   STATUS[676].EXT.BIT30 := FALSE;
   STATUS[676].EXT.BIT31 := FALSE;
   STATUS[676].EXT.ModeBit1 := FALSE;
   STATUS[676].EXT.ModeBit2 := FALSE;
   STATUS[676].EXT.ModeBit3 := FALSE;
   STATUS[676].EXT.BIT19 := FALSE;
   STATUS[676].EXT.BIT20 := FALSE;
   STATUS[676].EXT.AlarmSuppressed := FALSE;
   STATUS[676].EXT.AlarmPresent := FALSE;
   STATUS[676].EXT.AlarmFailUnAck := FALSE;
   STATUS[676].Status := 0;
   STATUS[676].TimeStamp := 16#0000;
   STATUS[677].EXT.AlarmWarnUnAck := FALSE;
   STATUS[677].EXT.AckRequired := FALSE;
   STATUS[677].EXT.Maintanence := FALSE;
   STATUS[677].EXT.Operation := FALSE;
   STATUS[677].EXT.Forced := FALSE;
   STATUS[677].EXT.BIT29 := FALSE;
   STATUS[677].EXT.BIT30 := FALSE;
   STATUS[677].EXT.BIT31 := FALSE;
   STATUS[677].EXT.ModeBit1 := FALSE;
   STATUS[677].EXT.ModeBit2 := FALSE;
   STATUS[677].EXT.ModeBit3 := FALSE;
   STATUS[677].EXT.BIT19 := FALSE;
   STATUS[677].EXT.BIT20 := FALSE;
   STATUS[677].EXT.AlarmSuppressed := FALSE;
   STATUS[677].EXT.AlarmPresent := FALSE;
   STATUS[677].EXT.AlarmFailUnAck := FALSE;
   STATUS[677].Status := 0;
   STATUS[677].TimeStamp := 16#0000;
   STATUS[678].EXT.AlarmWarnUnAck := FALSE;
   STATUS[678].EXT.AckRequired := FALSE;
   STATUS[678].EXT.Maintanence := FALSE;
   STATUS[678].EXT.Operation := FALSE;
   STATUS[678].EXT.Forced := FALSE;
   STATUS[678].EXT.BIT29 := FALSE;
   STATUS[678].EXT.BIT30 := FALSE;
   STATUS[678].EXT.BIT31 := FALSE;
   STATUS[678].EXT.ModeBit1 := FALSE;
   STATUS[678].EXT.ModeBit2 := FALSE;
   STATUS[678].EXT.ModeBit3 := FALSE;
   STATUS[678].EXT.BIT19 := FALSE;
   STATUS[678].EXT.BIT20 := FALSE;
   STATUS[678].EXT.AlarmSuppressed := FALSE;
   STATUS[678].EXT.AlarmPresent := FALSE;
   STATUS[678].EXT.AlarmFailUnAck := FALSE;
   STATUS[678].Status := 0;
   STATUS[678].TimeStamp := 16#0000;
   STATUS[679].EXT.AlarmWarnUnAck := FALSE;
   STATUS[679].EXT.AckRequired := FALSE;
   STATUS[679].EXT.Maintanence := FALSE;
   STATUS[679].EXT.Operation := FALSE;
   STATUS[679].EXT.Forced := FALSE;
   STATUS[679].EXT.BIT29 := FALSE;
   STATUS[679].EXT.BIT30 := FALSE;
   STATUS[679].EXT.BIT31 := FALSE;
   STATUS[679].EXT.ModeBit1 := FALSE;
   STATUS[679].EXT.ModeBit2 := FALSE;
   STATUS[679].EXT.ModeBit3 := FALSE;
   STATUS[679].EXT.BIT19 := FALSE;
   STATUS[679].EXT.BIT20 := FALSE;
   STATUS[679].EXT.AlarmSuppressed := FALSE;
   STATUS[679].EXT.AlarmPresent := FALSE;
   STATUS[679].EXT.AlarmFailUnAck := FALSE;
   STATUS[679].Status := 0;
   STATUS[679].TimeStamp := 16#0000;
   STATUS[680].EXT.AlarmWarnUnAck := FALSE;
   STATUS[680].EXT.AckRequired := FALSE;
   STATUS[680].EXT.Maintanence := FALSE;
   STATUS[680].EXT.Operation := FALSE;
   STATUS[680].EXT.Forced := FALSE;
   STATUS[680].EXT.BIT29 := FALSE;
   STATUS[680].EXT.BIT30 := FALSE;
   STATUS[680].EXT.BIT31 := FALSE;
   STATUS[680].EXT.ModeBit1 := FALSE;
   STATUS[680].EXT.ModeBit2 := FALSE;
   STATUS[680].EXT.ModeBit3 := FALSE;
   STATUS[680].EXT.BIT19 := FALSE;
   STATUS[680].EXT.BIT20 := FALSE;
   STATUS[680].EXT.AlarmSuppressed := FALSE;
   STATUS[680].EXT.AlarmPresent := FALSE;
   STATUS[680].EXT.AlarmFailUnAck := FALSE;
   STATUS[680].Status := 0;
   STATUS[680].TimeStamp := 16#0000;
   STATUS[681].EXT.AlarmWarnUnAck := FALSE;
   STATUS[681].EXT.AckRequired := FALSE;
   STATUS[681].EXT.Maintanence := FALSE;
   STATUS[681].EXT.Operation := FALSE;
   STATUS[681].EXT.Forced := FALSE;
   STATUS[681].EXT.BIT29 := FALSE;
   STATUS[681].EXT.BIT30 := FALSE;
   STATUS[681].EXT.BIT31 := FALSE;
   STATUS[681].EXT.ModeBit1 := FALSE;
   STATUS[681].EXT.ModeBit2 := FALSE;
   STATUS[681].EXT.ModeBit3 := FALSE;
   STATUS[681].EXT.BIT19 := FALSE;
   STATUS[681].EXT.BIT20 := FALSE;
   STATUS[681].EXT.AlarmSuppressed := FALSE;
   STATUS[681].EXT.AlarmPresent := FALSE;
   STATUS[681].EXT.AlarmFailUnAck := FALSE;
   STATUS[681].Status := 0;
   STATUS[681].TimeStamp := 16#0000;
   STATUS[682].EXT.AlarmWarnUnAck := FALSE;
   STATUS[682].EXT.AckRequired := FALSE;
   STATUS[682].EXT.Maintanence := FALSE;
   STATUS[682].EXT.Operation := FALSE;
   STATUS[682].EXT.Forced := FALSE;
   STATUS[682].EXT.BIT29 := FALSE;
   STATUS[682].EXT.BIT30 := FALSE;
   STATUS[682].EXT.BIT31 := FALSE;
   STATUS[682].EXT.ModeBit1 := FALSE;
   STATUS[682].EXT.ModeBit2 := FALSE;
   STATUS[682].EXT.ModeBit3 := FALSE;
   STATUS[682].EXT.BIT19 := FALSE;
   STATUS[682].EXT.BIT20 := FALSE;
   STATUS[682].EXT.AlarmSuppressed := FALSE;
   STATUS[682].EXT.AlarmPresent := FALSE;
   STATUS[682].EXT.AlarmFailUnAck := FALSE;
   STATUS[682].Status := 0;
   STATUS[682].TimeStamp := 16#0000;
   STATUS[683].EXT.AlarmWarnUnAck := FALSE;
   STATUS[683].EXT.AckRequired := FALSE;
   STATUS[683].EXT.Maintanence := FALSE;
   STATUS[683].EXT.Operation := FALSE;
   STATUS[683].EXT.Forced := FALSE;
   STATUS[683].EXT.BIT29 := FALSE;
   STATUS[683].EXT.BIT30 := FALSE;
   STATUS[683].EXT.BIT31 := FALSE;
   STATUS[683].EXT.ModeBit1 := FALSE;
   STATUS[683].EXT.ModeBit2 := FALSE;
   STATUS[683].EXT.ModeBit3 := FALSE;
   STATUS[683].EXT.BIT19 := FALSE;
   STATUS[683].EXT.BIT20 := FALSE;
   STATUS[683].EXT.AlarmSuppressed := FALSE;
   STATUS[683].EXT.AlarmPresent := FALSE;
   STATUS[683].EXT.AlarmFailUnAck := FALSE;
   STATUS[683].Status := 0;
   STATUS[683].TimeStamp := 16#0000;
   STATUS[684].EXT.AlarmWarnUnAck := FALSE;
   STATUS[684].EXT.AckRequired := FALSE;
   STATUS[684].EXT.Maintanence := FALSE;
   STATUS[684].EXT.Operation := FALSE;
   STATUS[684].EXT.Forced := FALSE;
   STATUS[684].EXT.BIT29 := FALSE;
   STATUS[684].EXT.BIT30 := FALSE;
   STATUS[684].EXT.BIT31 := FALSE;
   STATUS[684].EXT.ModeBit1 := FALSE;
   STATUS[684].EXT.ModeBit2 := FALSE;
   STATUS[684].EXT.ModeBit3 := FALSE;
   STATUS[684].EXT.BIT19 := FALSE;
   STATUS[684].EXT.BIT20 := FALSE;
   STATUS[684].EXT.AlarmSuppressed := FALSE;
   STATUS[684].EXT.AlarmPresent := FALSE;
   STATUS[684].EXT.AlarmFailUnAck := FALSE;
   STATUS[684].Status := 0;
   STATUS[684].TimeStamp := 16#0000;
   STATUS[685].EXT.AlarmWarnUnAck := FALSE;
   STATUS[685].EXT.AckRequired := FALSE;
   STATUS[685].EXT.Maintanence := FALSE;
   STATUS[685].EXT.Operation := FALSE;
   STATUS[685].EXT.Forced := FALSE;
   STATUS[685].EXT.BIT29 := FALSE;
   STATUS[685].EXT.BIT30 := FALSE;
   STATUS[685].EXT.BIT31 := FALSE;
   STATUS[685].EXT.ModeBit1 := FALSE;
   STATUS[685].EXT.ModeBit2 := FALSE;
   STATUS[685].EXT.ModeBit3 := FALSE;
   STATUS[685].EXT.BIT19 := FALSE;
   STATUS[685].EXT.BIT20 := FALSE;
   STATUS[685].EXT.AlarmSuppressed := FALSE;
   STATUS[685].EXT.AlarmPresent := FALSE;
   STATUS[685].EXT.AlarmFailUnAck := FALSE;
   STATUS[685].Status := 0;
   STATUS[685].TimeStamp := 16#0000;
   STATUS[686].EXT.AlarmWarnUnAck := FALSE;
   STATUS[686].EXT.AckRequired := FALSE;
   STATUS[686].EXT.Maintanence := FALSE;
   STATUS[686].EXT.Operation := FALSE;
   STATUS[686].EXT.Forced := FALSE;
   STATUS[686].EXT.BIT29 := FALSE;
   STATUS[686].EXT.BIT30 := FALSE;
   STATUS[686].EXT.BIT31 := FALSE;
   STATUS[686].EXT.ModeBit1 := FALSE;
   STATUS[686].EXT.ModeBit2 := FALSE;
   STATUS[686].EXT.ModeBit3 := FALSE;
   STATUS[686].EXT.BIT19 := FALSE;
   STATUS[686].EXT.BIT20 := FALSE;
   STATUS[686].EXT.AlarmSuppressed := FALSE;
   STATUS[686].EXT.AlarmPresent := FALSE;
   STATUS[686].EXT.AlarmFailUnAck := FALSE;
   STATUS[686].Status := 0;
   STATUS[686].TimeStamp := 16#0000;
   STATUS[687].EXT.AlarmWarnUnAck := FALSE;
   STATUS[687].EXT.AckRequired := FALSE;
   STATUS[687].EXT.Maintanence := FALSE;
   STATUS[687].EXT.Operation := FALSE;
   STATUS[687].EXT.Forced := FALSE;
   STATUS[687].EXT.BIT29 := FALSE;
   STATUS[687].EXT.BIT30 := FALSE;
   STATUS[687].EXT.BIT31 := FALSE;
   STATUS[687].EXT.ModeBit1 := FALSE;
   STATUS[687].EXT.ModeBit2 := FALSE;
   STATUS[687].EXT.ModeBit3 := FALSE;
   STATUS[687].EXT.BIT19 := FALSE;
   STATUS[687].EXT.BIT20 := FALSE;
   STATUS[687].EXT.AlarmSuppressed := FALSE;
   STATUS[687].EXT.AlarmPresent := FALSE;
   STATUS[687].EXT.AlarmFailUnAck := FALSE;
   STATUS[687].Status := 0;
   STATUS[687].TimeStamp := 16#0000;
   STATUS[688].EXT.AlarmWarnUnAck := FALSE;
   STATUS[688].EXT.AckRequired := FALSE;
   STATUS[688].EXT.Maintanence := FALSE;
   STATUS[688].EXT.Operation := FALSE;
   STATUS[688].EXT.Forced := FALSE;
   STATUS[688].EXT.BIT29 := FALSE;
   STATUS[688].EXT.BIT30 := FALSE;
   STATUS[688].EXT.BIT31 := FALSE;
   STATUS[688].EXT.ModeBit1 := FALSE;
   STATUS[688].EXT.ModeBit2 := FALSE;
   STATUS[688].EXT.ModeBit3 := FALSE;
   STATUS[688].EXT.BIT19 := FALSE;
   STATUS[688].EXT.BIT20 := FALSE;
   STATUS[688].EXT.AlarmSuppressed := FALSE;
   STATUS[688].EXT.AlarmPresent := FALSE;
   STATUS[688].EXT.AlarmFailUnAck := FALSE;
   STATUS[688].Status := 0;
   STATUS[688].TimeStamp := 16#0000;
   STATUS[689].EXT.AlarmWarnUnAck := FALSE;
   STATUS[689].EXT.AckRequired := FALSE;
   STATUS[689].EXT.Maintanence := FALSE;
   STATUS[689].EXT.Operation := FALSE;
   STATUS[689].EXT.Forced := FALSE;
   STATUS[689].EXT.BIT29 := FALSE;
   STATUS[689].EXT.BIT30 := FALSE;
   STATUS[689].EXT.BIT31 := FALSE;
   STATUS[689].EXT.ModeBit1 := FALSE;
   STATUS[689].EXT.ModeBit2 := FALSE;
   STATUS[689].EXT.ModeBit3 := FALSE;
   STATUS[689].EXT.BIT19 := FALSE;
   STATUS[689].EXT.BIT20 := FALSE;
   STATUS[689].EXT.AlarmSuppressed := FALSE;
   STATUS[689].EXT.AlarmPresent := FALSE;
   STATUS[689].EXT.AlarmFailUnAck := FALSE;
   STATUS[689].Status := 0;
   STATUS[689].TimeStamp := 16#0000;
   STATUS[690].EXT.AlarmWarnUnAck := FALSE;
   STATUS[690].EXT.AckRequired := FALSE;
   STATUS[690].EXT.Maintanence := FALSE;
   STATUS[690].EXT.Operation := FALSE;
   STATUS[690].EXT.Forced := FALSE;
   STATUS[690].EXT.BIT29 := FALSE;
   STATUS[690].EXT.BIT30 := FALSE;
   STATUS[690].EXT.BIT31 := FALSE;
   STATUS[690].EXT.ModeBit1 := FALSE;
   STATUS[690].EXT.ModeBit2 := FALSE;
   STATUS[690].EXT.ModeBit3 := FALSE;
   STATUS[690].EXT.BIT19 := FALSE;
   STATUS[690].EXT.BIT20 := FALSE;
   STATUS[690].EXT.AlarmSuppressed := FALSE;
   STATUS[690].EXT.AlarmPresent := FALSE;
   STATUS[690].EXT.AlarmFailUnAck := FALSE;
   STATUS[690].Status := 0;
   STATUS[690].TimeStamp := 16#0000;
   STATUS[691].EXT.AlarmWarnUnAck := FALSE;
   STATUS[691].EXT.AckRequired := FALSE;
   STATUS[691].EXT.Maintanence := FALSE;
   STATUS[691].EXT.Operation := FALSE;
   STATUS[691].EXT.Forced := FALSE;
   STATUS[691].EXT.BIT29 := FALSE;
   STATUS[691].EXT.BIT30 := FALSE;
   STATUS[691].EXT.BIT31 := FALSE;
   STATUS[691].EXT.ModeBit1 := FALSE;
   STATUS[691].EXT.ModeBit2 := FALSE;
   STATUS[691].EXT.ModeBit3 := FALSE;
   STATUS[691].EXT.BIT19 := FALSE;
   STATUS[691].EXT.BIT20 := FALSE;
   STATUS[691].EXT.AlarmSuppressed := FALSE;
   STATUS[691].EXT.AlarmPresent := FALSE;
   STATUS[691].EXT.AlarmFailUnAck := FALSE;
   STATUS[691].Status := 0;
   STATUS[691].TimeStamp := 16#0000;
   STATUS[692].EXT.AlarmWarnUnAck := FALSE;
   STATUS[692].EXT.AckRequired := FALSE;
   STATUS[692].EXT.Maintanence := FALSE;
   STATUS[692].EXT.Operation := FALSE;
   STATUS[692].EXT.Forced := FALSE;
   STATUS[692].EXT.BIT29 := FALSE;
   STATUS[692].EXT.BIT30 := FALSE;
   STATUS[692].EXT.BIT31 := FALSE;
   STATUS[692].EXT.ModeBit1 := FALSE;
   STATUS[692].EXT.ModeBit2 := FALSE;
   STATUS[692].EXT.ModeBit3 := FALSE;
   STATUS[692].EXT.BIT19 := FALSE;
   STATUS[692].EXT.BIT20 := FALSE;
   STATUS[692].EXT.AlarmSuppressed := FALSE;
   STATUS[692].EXT.AlarmPresent := FALSE;
   STATUS[692].EXT.AlarmFailUnAck := FALSE;
   STATUS[692].Status := 0;
   STATUS[692].TimeStamp := 16#0000;
   STATUS[693].EXT.AlarmWarnUnAck := FALSE;
   STATUS[693].EXT.AckRequired := FALSE;
   STATUS[693].EXT.Maintanence := FALSE;
   STATUS[693].EXT.Operation := FALSE;
   STATUS[693].EXT.Forced := FALSE;
   STATUS[693].EXT.BIT29 := FALSE;
   STATUS[693].EXT.BIT30 := FALSE;
   STATUS[693].EXT.BIT31 := FALSE;
   STATUS[693].EXT.ModeBit1 := FALSE;
   STATUS[693].EXT.ModeBit2 := FALSE;
   STATUS[693].EXT.ModeBit3 := FALSE;
   STATUS[693].EXT.BIT19 := FALSE;
   STATUS[693].EXT.BIT20 := FALSE;
   STATUS[693].EXT.AlarmSuppressed := FALSE;
   STATUS[693].EXT.AlarmPresent := FALSE;
   STATUS[693].EXT.AlarmFailUnAck := FALSE;
   STATUS[693].Status := 0;
   STATUS[693].TimeStamp := 16#0000;
   STATUS[694].EXT.AlarmWarnUnAck := FALSE;
   STATUS[694].EXT.AckRequired := FALSE;
   STATUS[694].EXT.Maintanence := FALSE;
   STATUS[694].EXT.Operation := FALSE;
   STATUS[694].EXT.Forced := FALSE;
   STATUS[694].EXT.BIT29 := FALSE;
   STATUS[694].EXT.BIT30 := FALSE;
   STATUS[694].EXT.BIT31 := FALSE;
   STATUS[694].EXT.ModeBit1 := FALSE;
   STATUS[694].EXT.ModeBit2 := FALSE;
   STATUS[694].EXT.ModeBit3 := FALSE;
   STATUS[694].EXT.BIT19 := FALSE;
   STATUS[694].EXT.BIT20 := FALSE;
   STATUS[694].EXT.AlarmSuppressed := FALSE;
   STATUS[694].EXT.AlarmPresent := FALSE;
   STATUS[694].EXT.AlarmFailUnAck := FALSE;
   STATUS[694].Status := 0;
   STATUS[694].TimeStamp := 16#0000;
   STATUS[695].EXT.AlarmWarnUnAck := FALSE;
   STATUS[695].EXT.AckRequired := FALSE;
   STATUS[695].EXT.Maintanence := FALSE;
   STATUS[695].EXT.Operation := FALSE;
   STATUS[695].EXT.Forced := FALSE;
   STATUS[695].EXT.BIT29 := FALSE;
   STATUS[695].EXT.BIT30 := FALSE;
   STATUS[695].EXT.BIT31 := FALSE;
   STATUS[695].EXT.ModeBit1 := FALSE;
   STATUS[695].EXT.ModeBit2 := FALSE;
   STATUS[695].EXT.ModeBit3 := FALSE;
   STATUS[695].EXT.BIT19 := FALSE;
   STATUS[695].EXT.BIT20 := FALSE;
   STATUS[695].EXT.AlarmSuppressed := FALSE;
   STATUS[695].EXT.AlarmPresent := FALSE;
   STATUS[695].EXT.AlarmFailUnAck := FALSE;
   STATUS[695].Status := 0;
   STATUS[695].TimeStamp := 16#0000;
   STATUS[696].EXT.AlarmWarnUnAck := FALSE;
   STATUS[696].EXT.AckRequired := FALSE;
   STATUS[696].EXT.Maintanence := FALSE;
   STATUS[696].EXT.Operation := FALSE;
   STATUS[696].EXT.Forced := FALSE;
   STATUS[696].EXT.BIT29 := FALSE;
   STATUS[696].EXT.BIT30 := FALSE;
   STATUS[696].EXT.BIT31 := FALSE;
   STATUS[696].EXT.ModeBit1 := FALSE;
   STATUS[696].EXT.ModeBit2 := FALSE;
   STATUS[696].EXT.ModeBit3 := FALSE;
   STATUS[696].EXT.BIT19 := FALSE;
   STATUS[696].EXT.BIT20 := FALSE;
   STATUS[696].EXT.AlarmSuppressed := FALSE;
   STATUS[696].EXT.AlarmPresent := FALSE;
   STATUS[696].EXT.AlarmFailUnAck := FALSE;
   STATUS[696].Status := 0;
   STATUS[696].TimeStamp := 16#0000;
   STATUS[697].EXT.AlarmWarnUnAck := FALSE;
   STATUS[697].EXT.AckRequired := FALSE;
   STATUS[697].EXT.Maintanence := FALSE;
   STATUS[697].EXT.Operation := FALSE;
   STATUS[697].EXT.Forced := FALSE;
   STATUS[697].EXT.BIT29 := FALSE;
   STATUS[697].EXT.BIT30 := FALSE;
   STATUS[697].EXT.BIT31 := FALSE;
   STATUS[697].EXT.ModeBit1 := FALSE;
   STATUS[697].EXT.ModeBit2 := FALSE;
   STATUS[697].EXT.ModeBit3 := FALSE;
   STATUS[697].EXT.BIT19 := FALSE;
   STATUS[697].EXT.BIT20 := FALSE;
   STATUS[697].EXT.AlarmSuppressed := FALSE;
   STATUS[697].EXT.AlarmPresent := FALSE;
   STATUS[697].EXT.AlarmFailUnAck := FALSE;
   STATUS[697].Status := 0;
   STATUS[697].TimeStamp := 16#0000;
   STATUS[698].EXT.AlarmWarnUnAck := FALSE;
   STATUS[698].EXT.AckRequired := FALSE;
   STATUS[698].EXT.Maintanence := FALSE;
   STATUS[698].EXT.Operation := FALSE;
   STATUS[698].EXT.Forced := FALSE;
   STATUS[698].EXT.BIT29 := FALSE;
   STATUS[698].EXT.BIT30 := FALSE;
   STATUS[698].EXT.BIT31 := FALSE;
   STATUS[698].EXT.ModeBit1 := FALSE;
   STATUS[698].EXT.ModeBit2 := FALSE;
   STATUS[698].EXT.ModeBit3 := FALSE;
   STATUS[698].EXT.BIT19 := FALSE;
   STATUS[698].EXT.BIT20 := FALSE;
   STATUS[698].EXT.AlarmSuppressed := FALSE;
   STATUS[698].EXT.AlarmPresent := FALSE;
   STATUS[698].EXT.AlarmFailUnAck := FALSE;
   STATUS[698].Status := 0;
   STATUS[698].TimeStamp := 16#0000;
   STATUS[699].EXT.AlarmWarnUnAck := FALSE;
   STATUS[699].EXT.AckRequired := FALSE;
   STATUS[699].EXT.Maintanence := FALSE;
   STATUS[699].EXT.Operation := FALSE;
   STATUS[699].EXT.Forced := FALSE;
   STATUS[699].EXT.BIT29 := FALSE;
   STATUS[699].EXT.BIT30 := FALSE;
   STATUS[699].EXT.BIT31 := FALSE;
   STATUS[699].EXT.ModeBit1 := FALSE;
   STATUS[699].EXT.ModeBit2 := FALSE;
   STATUS[699].EXT.ModeBit3 := FALSE;
   STATUS[699].EXT.BIT19 := FALSE;
   STATUS[699].EXT.BIT20 := FALSE;
   STATUS[699].EXT.AlarmSuppressed := FALSE;
   STATUS[699].EXT.AlarmPresent := FALSE;
   STATUS[699].EXT.AlarmFailUnAck := FALSE;
   STATUS[699].Status := 0;
   STATUS[699].TimeStamp := 16#0000;
   STATUS[700].EXT.AlarmWarnUnAck := FALSE;
   STATUS[700].EXT.AckRequired := FALSE;
   STATUS[700].EXT.Maintanence := FALSE;
   STATUS[700].EXT.Operation := FALSE;
   STATUS[700].EXT.Forced := FALSE;
   STATUS[700].EXT.BIT29 := FALSE;
   STATUS[700].EXT.BIT30 := FALSE;
   STATUS[700].EXT.BIT31 := FALSE;
   STATUS[700].EXT.ModeBit1 := FALSE;
   STATUS[700].EXT.ModeBit2 := FALSE;
   STATUS[700].EXT.ModeBit3 := FALSE;
   STATUS[700].EXT.BIT19 := FALSE;
   STATUS[700].EXT.BIT20 := FALSE;
   STATUS[700].EXT.AlarmSuppressed := FALSE;
   STATUS[700].EXT.AlarmPresent := FALSE;
   STATUS[700].EXT.AlarmFailUnAck := FALSE;
   STATUS[700].Status := 0;
   STATUS[700].TimeStamp := 16#0000;
   STATUS[701].EXT.AlarmWarnUnAck := FALSE;
   STATUS[701].EXT.AckRequired := FALSE;
   STATUS[701].EXT.Maintanence := FALSE;
   STATUS[701].EXT.Operation := FALSE;
   STATUS[701].EXT.Forced := FALSE;
   STATUS[701].EXT.BIT29 := FALSE;
   STATUS[701].EXT.BIT30 := FALSE;
   STATUS[701].EXT.BIT31 := FALSE;
   STATUS[701].EXT.ModeBit1 := FALSE;
   STATUS[701].EXT.ModeBit2 := FALSE;
   STATUS[701].EXT.ModeBit3 := FALSE;
   STATUS[701].EXT.BIT19 := FALSE;
   STATUS[701].EXT.BIT20 := FALSE;
   STATUS[701].EXT.AlarmSuppressed := FALSE;
   STATUS[701].EXT.AlarmPresent := FALSE;
   STATUS[701].EXT.AlarmFailUnAck := FALSE;
   STATUS[701].Status := 0;
   STATUS[701].TimeStamp := 16#0000;
   STATUS[702].EXT.AlarmWarnUnAck := FALSE;
   STATUS[702].EXT.AckRequired := FALSE;
   STATUS[702].EXT.Maintanence := FALSE;
   STATUS[702].EXT.Operation := FALSE;
   STATUS[702].EXT.Forced := FALSE;
   STATUS[702].EXT.BIT29 := FALSE;
   STATUS[702].EXT.BIT30 := FALSE;
   STATUS[702].EXT.BIT31 := FALSE;
   STATUS[702].EXT.ModeBit1 := FALSE;
   STATUS[702].EXT.ModeBit2 := FALSE;
   STATUS[702].EXT.ModeBit3 := FALSE;
   STATUS[702].EXT.BIT19 := FALSE;
   STATUS[702].EXT.BIT20 := FALSE;
   STATUS[702].EXT.AlarmSuppressed := FALSE;
   STATUS[702].EXT.AlarmPresent := FALSE;
   STATUS[702].EXT.AlarmFailUnAck := FALSE;
   STATUS[702].Status := 0;
   STATUS[702].TimeStamp := 16#0000;
   STATUS[703].EXT.AlarmWarnUnAck := FALSE;
   STATUS[703].EXT.AckRequired := FALSE;
   STATUS[703].EXT.Maintanence := FALSE;
   STATUS[703].EXT.Operation := FALSE;
   STATUS[703].EXT.Forced := FALSE;
   STATUS[703].EXT.BIT29 := FALSE;
   STATUS[703].EXT.BIT30 := FALSE;
   STATUS[703].EXT.BIT31 := FALSE;
   STATUS[703].EXT.ModeBit1 := FALSE;
   STATUS[703].EXT.ModeBit2 := FALSE;
   STATUS[703].EXT.ModeBit3 := FALSE;
   STATUS[703].EXT.BIT19 := FALSE;
   STATUS[703].EXT.BIT20 := FALSE;
   STATUS[703].EXT.AlarmSuppressed := FALSE;
   STATUS[703].EXT.AlarmPresent := FALSE;
   STATUS[703].EXT.AlarmFailUnAck := FALSE;
   STATUS[703].Status := 0;
   STATUS[703].TimeStamp := 16#0000;
   STATUS[704].EXT.AlarmWarnUnAck := FALSE;
   STATUS[704].EXT.AckRequired := FALSE;
   STATUS[704].EXT.Maintanence := FALSE;
   STATUS[704].EXT.Operation := FALSE;
   STATUS[704].EXT.Forced := FALSE;
   STATUS[704].EXT.BIT29 := FALSE;
   STATUS[704].EXT.BIT30 := FALSE;
   STATUS[704].EXT.BIT31 := FALSE;
   STATUS[704].EXT.ModeBit1 := FALSE;
   STATUS[704].EXT.ModeBit2 := FALSE;
   STATUS[704].EXT.ModeBit3 := FALSE;
   STATUS[704].EXT.BIT19 := FALSE;
   STATUS[704].EXT.BIT20 := FALSE;
   STATUS[704].EXT.AlarmSuppressed := FALSE;
   STATUS[704].EXT.AlarmPresent := FALSE;
   STATUS[704].EXT.AlarmFailUnAck := FALSE;
   STATUS[704].Status := 0;
   STATUS[704].TimeStamp := 16#0000;
   STATUS[705].EXT.AlarmWarnUnAck := FALSE;
   STATUS[705].EXT.AckRequired := FALSE;
   STATUS[705].EXT.Maintanence := FALSE;
   STATUS[705].EXT.Operation := FALSE;
   STATUS[705].EXT.Forced := FALSE;
   STATUS[705].EXT.BIT29 := FALSE;
   STATUS[705].EXT.BIT30 := FALSE;
   STATUS[705].EXT.BIT31 := FALSE;
   STATUS[705].EXT.ModeBit1 := FALSE;
   STATUS[705].EXT.ModeBit2 := FALSE;
   STATUS[705].EXT.ModeBit3 := FALSE;
   STATUS[705].EXT.BIT19 := FALSE;
   STATUS[705].EXT.BIT20 := FALSE;
   STATUS[705].EXT.AlarmSuppressed := FALSE;
   STATUS[705].EXT.AlarmPresent := FALSE;
   STATUS[705].EXT.AlarmFailUnAck := FALSE;
   STATUS[705].Status := 0;
   STATUS[705].TimeStamp := 16#0000;
   STATUS[706].EXT.AlarmWarnUnAck := FALSE;
   STATUS[706].EXT.AckRequired := FALSE;
   STATUS[706].EXT.Maintanence := FALSE;
   STATUS[706].EXT.Operation := FALSE;
   STATUS[706].EXT.Forced := FALSE;
   STATUS[706].EXT.BIT29 := FALSE;
   STATUS[706].EXT.BIT30 := FALSE;
   STATUS[706].EXT.BIT31 := FALSE;
   STATUS[706].EXT.ModeBit1 := FALSE;
   STATUS[706].EXT.ModeBit2 := FALSE;
   STATUS[706].EXT.ModeBit3 := FALSE;
   STATUS[706].EXT.BIT19 := FALSE;
   STATUS[706].EXT.BIT20 := FALSE;
   STATUS[706].EXT.AlarmSuppressed := FALSE;
   STATUS[706].EXT.AlarmPresent := FALSE;
   STATUS[706].EXT.AlarmFailUnAck := FALSE;
   STATUS[706].Status := 0;
   STATUS[706].TimeStamp := 16#0000;
   STATUS[707].EXT.AlarmWarnUnAck := FALSE;
   STATUS[707].EXT.AckRequired := FALSE;
   STATUS[707].EXT.Maintanence := FALSE;
   STATUS[707].EXT.Operation := FALSE;
   STATUS[707].EXT.Forced := FALSE;
   STATUS[707].EXT.BIT29 := FALSE;
   STATUS[707].EXT.BIT30 := FALSE;
   STATUS[707].EXT.BIT31 := FALSE;
   STATUS[707].EXT.ModeBit1 := FALSE;
   STATUS[707].EXT.ModeBit2 := FALSE;
   STATUS[707].EXT.ModeBit3 := FALSE;
   STATUS[707].EXT.BIT19 := FALSE;
   STATUS[707].EXT.BIT20 := FALSE;
   STATUS[707].EXT.AlarmSuppressed := FALSE;
   STATUS[707].EXT.AlarmPresent := FALSE;
   STATUS[707].EXT.AlarmFailUnAck := FALSE;
   STATUS[707].Status := 0;
   STATUS[707].TimeStamp := 16#0000;
   STATUS[708].EXT.AlarmWarnUnAck := FALSE;
   STATUS[708].EXT.AckRequired := FALSE;
   STATUS[708].EXT.Maintanence := FALSE;
   STATUS[708].EXT.Operation := FALSE;
   STATUS[708].EXT.Forced := FALSE;
   STATUS[708].EXT.BIT29 := FALSE;
   STATUS[708].EXT.BIT30 := FALSE;
   STATUS[708].EXT.BIT31 := FALSE;
   STATUS[708].EXT.ModeBit1 := FALSE;
   STATUS[708].EXT.ModeBit2 := FALSE;
   STATUS[708].EXT.ModeBit3 := FALSE;
   STATUS[708].EXT.BIT19 := FALSE;
   STATUS[708].EXT.BIT20 := FALSE;
   STATUS[708].EXT.AlarmSuppressed := FALSE;
   STATUS[708].EXT.AlarmPresent := FALSE;
   STATUS[708].EXT.AlarmFailUnAck := FALSE;
   STATUS[708].Status := 0;
   STATUS[708].TimeStamp := 16#0000;
   STATUS[709].EXT.AlarmWarnUnAck := FALSE;
   STATUS[709].EXT.AckRequired := FALSE;
   STATUS[709].EXT.Maintanence := FALSE;
   STATUS[709].EXT.Operation := FALSE;
   STATUS[709].EXT.Forced := FALSE;
   STATUS[709].EXT.BIT29 := FALSE;
   STATUS[709].EXT.BIT30 := FALSE;
   STATUS[709].EXT.BIT31 := FALSE;
   STATUS[709].EXT.ModeBit1 := FALSE;
   STATUS[709].EXT.ModeBit2 := FALSE;
   STATUS[709].EXT.ModeBit3 := FALSE;
   STATUS[709].EXT.BIT19 := FALSE;
   STATUS[709].EXT.BIT20 := FALSE;
   STATUS[709].EXT.AlarmSuppressed := FALSE;
   STATUS[709].EXT.AlarmPresent := FALSE;
   STATUS[709].EXT.AlarmFailUnAck := FALSE;
   STATUS[709].Status := 0;
   STATUS[709].TimeStamp := 16#0000;
   STATUS[710].EXT.AlarmWarnUnAck := FALSE;
   STATUS[710].EXT.AckRequired := FALSE;
   STATUS[710].EXT.Maintanence := FALSE;
   STATUS[710].EXT.Operation := FALSE;
   STATUS[710].EXT.Forced := FALSE;
   STATUS[710].EXT.BIT29 := FALSE;
   STATUS[710].EXT.BIT30 := FALSE;
   STATUS[710].EXT.BIT31 := FALSE;
   STATUS[710].EXT.ModeBit1 := FALSE;
   STATUS[710].EXT.ModeBit2 := FALSE;
   STATUS[710].EXT.ModeBit3 := FALSE;
   STATUS[710].EXT.BIT19 := FALSE;
   STATUS[710].EXT.BIT20 := FALSE;
   STATUS[710].EXT.AlarmSuppressed := FALSE;
   STATUS[710].EXT.AlarmPresent := FALSE;
   STATUS[710].EXT.AlarmFailUnAck := FALSE;
   STATUS[710].Status := 0;
   STATUS[710].TimeStamp := 16#0000;
   STATUS[711].EXT.AlarmWarnUnAck := FALSE;
   STATUS[711].EXT.AckRequired := FALSE;
   STATUS[711].EXT.Maintanence := FALSE;
   STATUS[711].EXT.Operation := FALSE;
   STATUS[711].EXT.Forced := FALSE;
   STATUS[711].EXT.BIT29 := FALSE;
   STATUS[711].EXT.BIT30 := FALSE;
   STATUS[711].EXT.BIT31 := FALSE;
   STATUS[711].EXT.ModeBit1 := FALSE;
   STATUS[711].EXT.ModeBit2 := FALSE;
   STATUS[711].EXT.ModeBit3 := FALSE;
   STATUS[711].EXT.BIT19 := FALSE;
   STATUS[711].EXT.BIT20 := FALSE;
   STATUS[711].EXT.AlarmSuppressed := FALSE;
   STATUS[711].EXT.AlarmPresent := FALSE;
   STATUS[711].EXT.AlarmFailUnAck := FALSE;
   STATUS[711].Status := 0;
   STATUS[711].TimeStamp := 16#0000;
   STATUS[712].EXT.AlarmWarnUnAck := FALSE;
   STATUS[712].EXT.AckRequired := FALSE;
   STATUS[712].EXT.Maintanence := FALSE;
   STATUS[712].EXT.Operation := FALSE;
   STATUS[712].EXT.Forced := FALSE;
   STATUS[712].EXT.BIT29 := FALSE;
   STATUS[712].EXT.BIT30 := FALSE;
   STATUS[712].EXT.BIT31 := FALSE;
   STATUS[712].EXT.ModeBit1 := FALSE;
   STATUS[712].EXT.ModeBit2 := FALSE;
   STATUS[712].EXT.ModeBit3 := FALSE;
   STATUS[712].EXT.BIT19 := FALSE;
   STATUS[712].EXT.BIT20 := FALSE;
   STATUS[712].EXT.AlarmSuppressed := FALSE;
   STATUS[712].EXT.AlarmPresent := FALSE;
   STATUS[712].EXT.AlarmFailUnAck := FALSE;
   STATUS[712].Status := 0;
   STATUS[712].TimeStamp := 16#0000;
   STATUS[713].EXT.AlarmWarnUnAck := FALSE;
   STATUS[713].EXT.AckRequired := FALSE;
   STATUS[713].EXT.Maintanence := FALSE;
   STATUS[713].EXT.Operation := FALSE;
   STATUS[713].EXT.Forced := FALSE;
   STATUS[713].EXT.BIT29 := FALSE;
   STATUS[713].EXT.BIT30 := FALSE;
   STATUS[713].EXT.BIT31 := FALSE;
   STATUS[713].EXT.ModeBit1 := FALSE;
   STATUS[713].EXT.ModeBit2 := FALSE;
   STATUS[713].EXT.ModeBit3 := FALSE;
   STATUS[713].EXT.BIT19 := FALSE;
   STATUS[713].EXT.BIT20 := FALSE;
   STATUS[713].EXT.AlarmSuppressed := FALSE;
   STATUS[713].EXT.AlarmPresent := FALSE;
   STATUS[713].EXT.AlarmFailUnAck := FALSE;
   STATUS[713].Status := 0;
   STATUS[713].TimeStamp := 16#0000;
   STATUS[714].EXT.AlarmWarnUnAck := FALSE;
   STATUS[714].EXT.AckRequired := FALSE;
   STATUS[714].EXT.Maintanence := FALSE;
   STATUS[714].EXT.Operation := FALSE;
   STATUS[714].EXT.Forced := FALSE;
   STATUS[714].EXT.BIT29 := FALSE;
   STATUS[714].EXT.BIT30 := FALSE;
   STATUS[714].EXT.BIT31 := FALSE;
   STATUS[714].EXT.ModeBit1 := FALSE;
   STATUS[714].EXT.ModeBit2 := FALSE;
   STATUS[714].EXT.ModeBit3 := FALSE;
   STATUS[714].EXT.BIT19 := FALSE;
   STATUS[714].EXT.BIT20 := FALSE;
   STATUS[714].EXT.AlarmSuppressed := FALSE;
   STATUS[714].EXT.AlarmPresent := FALSE;
   STATUS[714].EXT.AlarmFailUnAck := FALSE;
   STATUS[714].Status := 0;
   STATUS[714].TimeStamp := 16#0000;
   STATUS[715].EXT.AlarmWarnUnAck := FALSE;
   STATUS[715].EXT.AckRequired := FALSE;
   STATUS[715].EXT.Maintanence := FALSE;
   STATUS[715].EXT.Operation := FALSE;
   STATUS[715].EXT.Forced := FALSE;
   STATUS[715].EXT.BIT29 := FALSE;
   STATUS[715].EXT.BIT30 := FALSE;
   STATUS[715].EXT.BIT31 := FALSE;
   STATUS[715].EXT.ModeBit1 := FALSE;
   STATUS[715].EXT.ModeBit2 := FALSE;
   STATUS[715].EXT.ModeBit3 := FALSE;
   STATUS[715].EXT.BIT19 := FALSE;
   STATUS[715].EXT.BIT20 := FALSE;
   STATUS[715].EXT.AlarmSuppressed := FALSE;
   STATUS[715].EXT.AlarmPresent := FALSE;
   STATUS[715].EXT.AlarmFailUnAck := FALSE;
   STATUS[715].Status := 0;
   STATUS[715].TimeStamp := 16#0000;
   STATUS[716].EXT.AlarmWarnUnAck := FALSE;
   STATUS[716].EXT.AckRequired := FALSE;
   STATUS[716].EXT.Maintanence := FALSE;
   STATUS[716].EXT.Operation := FALSE;
   STATUS[716].EXT.Forced := FALSE;
   STATUS[716].EXT.BIT29 := FALSE;
   STATUS[716].EXT.BIT30 := FALSE;
   STATUS[716].EXT.BIT31 := FALSE;
   STATUS[716].EXT.ModeBit1 := FALSE;
   STATUS[716].EXT.ModeBit2 := FALSE;
   STATUS[716].EXT.ModeBit3 := FALSE;
   STATUS[716].EXT.BIT19 := FALSE;
   STATUS[716].EXT.BIT20 := FALSE;
   STATUS[716].EXT.AlarmSuppressed := FALSE;
   STATUS[716].EXT.AlarmPresent := FALSE;
   STATUS[716].EXT.AlarmFailUnAck := FALSE;
   STATUS[716].Status := 0;
   STATUS[716].TimeStamp := 16#0000;
   STATUS[717].EXT.AlarmWarnUnAck := FALSE;
   STATUS[717].EXT.AckRequired := FALSE;
   STATUS[717].EXT.Maintanence := FALSE;
   STATUS[717].EXT.Operation := FALSE;
   STATUS[717].EXT.Forced := FALSE;
   STATUS[717].EXT.BIT29 := FALSE;
   STATUS[717].EXT.BIT30 := FALSE;
   STATUS[717].EXT.BIT31 := FALSE;
   STATUS[717].EXT.ModeBit1 := FALSE;
   STATUS[717].EXT.ModeBit2 := FALSE;
   STATUS[717].EXT.ModeBit3 := FALSE;
   STATUS[717].EXT.BIT19 := FALSE;
   STATUS[717].EXT.BIT20 := FALSE;
   STATUS[717].EXT.AlarmSuppressed := FALSE;
   STATUS[717].EXT.AlarmPresent := FALSE;
   STATUS[717].EXT.AlarmFailUnAck := FALSE;
   STATUS[717].Status := 0;
   STATUS[717].TimeStamp := 16#0000;
   STATUS[718].EXT.AlarmWarnUnAck := FALSE;
   STATUS[718].EXT.AckRequired := FALSE;
   STATUS[718].EXT.Maintanence := FALSE;
   STATUS[718].EXT.Operation := FALSE;
   STATUS[718].EXT.Forced := FALSE;
   STATUS[718].EXT.BIT29 := FALSE;
   STATUS[718].EXT.BIT30 := FALSE;
   STATUS[718].EXT.BIT31 := FALSE;
   STATUS[718].EXT.ModeBit1 := FALSE;
   STATUS[718].EXT.ModeBit2 := FALSE;
   STATUS[718].EXT.ModeBit3 := FALSE;
   STATUS[718].EXT.BIT19 := FALSE;
   STATUS[718].EXT.BIT20 := FALSE;
   STATUS[718].EXT.AlarmSuppressed := FALSE;
   STATUS[718].EXT.AlarmPresent := FALSE;
   STATUS[718].EXT.AlarmFailUnAck := FALSE;
   STATUS[718].Status := 0;
   STATUS[718].TimeStamp := 16#0000;
   STATUS[719].EXT.AlarmWarnUnAck := FALSE;
   STATUS[719].EXT.AckRequired := FALSE;
   STATUS[719].EXT.Maintanence := FALSE;
   STATUS[719].EXT.Operation := FALSE;
   STATUS[719].EXT.Forced := FALSE;
   STATUS[719].EXT.BIT29 := FALSE;
   STATUS[719].EXT.BIT30 := FALSE;
   STATUS[719].EXT.BIT31 := FALSE;
   STATUS[719].EXT.ModeBit1 := FALSE;
   STATUS[719].EXT.ModeBit2 := FALSE;
   STATUS[719].EXT.ModeBit3 := FALSE;
   STATUS[719].EXT.BIT19 := FALSE;
   STATUS[719].EXT.BIT20 := FALSE;
   STATUS[719].EXT.AlarmSuppressed := FALSE;
   STATUS[719].EXT.AlarmPresent := FALSE;
   STATUS[719].EXT.AlarmFailUnAck := FALSE;
   STATUS[719].Status := 0;
   STATUS[719].TimeStamp := 16#0000;
   STATUS[720].EXT.AlarmWarnUnAck := FALSE;
   STATUS[720].EXT.AckRequired := FALSE;
   STATUS[720].EXT.Maintanence := FALSE;
   STATUS[720].EXT.Operation := FALSE;
   STATUS[720].EXT.Forced := FALSE;
   STATUS[720].EXT.BIT29 := FALSE;
   STATUS[720].EXT.BIT30 := FALSE;
   STATUS[720].EXT.BIT31 := FALSE;
   STATUS[720].EXT.ModeBit1 := FALSE;
   STATUS[720].EXT.ModeBit2 := FALSE;
   STATUS[720].EXT.ModeBit3 := FALSE;
   STATUS[720].EXT.BIT19 := FALSE;
   STATUS[720].EXT.BIT20 := FALSE;
   STATUS[720].EXT.AlarmSuppressed := FALSE;
   STATUS[720].EXT.AlarmPresent := FALSE;
   STATUS[720].EXT.AlarmFailUnAck := FALSE;
   STATUS[720].Status := 0;
   STATUS[720].TimeStamp := 16#0000;
   STATUS[721].EXT.AlarmWarnUnAck := FALSE;
   STATUS[721].EXT.AckRequired := FALSE;
   STATUS[721].EXT.Maintanence := FALSE;
   STATUS[721].EXT.Operation := FALSE;
   STATUS[721].EXT.Forced := FALSE;
   STATUS[721].EXT.BIT29 := FALSE;
   STATUS[721].EXT.BIT30 := FALSE;
   STATUS[721].EXT.BIT31 := FALSE;
   STATUS[721].EXT.ModeBit1 := FALSE;
   STATUS[721].EXT.ModeBit2 := FALSE;
   STATUS[721].EXT.ModeBit3 := FALSE;
   STATUS[721].EXT.BIT19 := FALSE;
   STATUS[721].EXT.BIT20 := FALSE;
   STATUS[721].EXT.AlarmSuppressed := FALSE;
   STATUS[721].EXT.AlarmPresent := FALSE;
   STATUS[721].EXT.AlarmFailUnAck := FALSE;
   STATUS[721].Status := 0;
   STATUS[721].TimeStamp := 16#0000;
   STATUS[722].EXT.AlarmWarnUnAck := FALSE;
   STATUS[722].EXT.AckRequired := FALSE;
   STATUS[722].EXT.Maintanence := FALSE;
   STATUS[722].EXT.Operation := FALSE;
   STATUS[722].EXT.Forced := FALSE;
   STATUS[722].EXT.BIT29 := FALSE;
   STATUS[722].EXT.BIT30 := FALSE;
   STATUS[722].EXT.BIT31 := FALSE;
   STATUS[722].EXT.ModeBit1 := FALSE;
   STATUS[722].EXT.ModeBit2 := FALSE;
   STATUS[722].EXT.ModeBit3 := FALSE;
   STATUS[722].EXT.BIT19 := FALSE;
   STATUS[722].EXT.BIT20 := FALSE;
   STATUS[722].EXT.AlarmSuppressed := FALSE;
   STATUS[722].EXT.AlarmPresent := FALSE;
   STATUS[722].EXT.AlarmFailUnAck := FALSE;
   STATUS[722].Status := 0;
   STATUS[722].TimeStamp := 16#0000;
   STATUS[723].EXT.AlarmWarnUnAck := FALSE;
   STATUS[723].EXT.AckRequired := FALSE;
   STATUS[723].EXT.Maintanence := FALSE;
   STATUS[723].EXT.Operation := FALSE;
   STATUS[723].EXT.Forced := FALSE;
   STATUS[723].EXT.BIT29 := FALSE;
   STATUS[723].EXT.BIT30 := FALSE;
   STATUS[723].EXT.BIT31 := FALSE;
   STATUS[723].EXT.ModeBit1 := FALSE;
   STATUS[723].EXT.ModeBit2 := FALSE;
   STATUS[723].EXT.ModeBit3 := FALSE;
   STATUS[723].EXT.BIT19 := FALSE;
   STATUS[723].EXT.BIT20 := FALSE;
   STATUS[723].EXT.AlarmSuppressed := FALSE;
   STATUS[723].EXT.AlarmPresent := FALSE;
   STATUS[723].EXT.AlarmFailUnAck := FALSE;
   STATUS[723].Status := 0;
   STATUS[723].TimeStamp := 16#0000;
   STATUS[724].EXT.AlarmWarnUnAck := FALSE;
   STATUS[724].EXT.AckRequired := FALSE;
   STATUS[724].EXT.Maintanence := FALSE;
   STATUS[724].EXT.Operation := FALSE;
   STATUS[724].EXT.Forced := FALSE;
   STATUS[724].EXT.BIT29 := FALSE;
   STATUS[724].EXT.BIT30 := FALSE;
   STATUS[724].EXT.BIT31 := FALSE;
   STATUS[724].EXT.ModeBit1 := FALSE;
   STATUS[724].EXT.ModeBit2 := FALSE;
   STATUS[724].EXT.ModeBit3 := FALSE;
   STATUS[724].EXT.BIT19 := FALSE;
   STATUS[724].EXT.BIT20 := FALSE;
   STATUS[724].EXT.AlarmSuppressed := FALSE;
   STATUS[724].EXT.AlarmPresent := FALSE;
   STATUS[724].EXT.AlarmFailUnAck := FALSE;
   STATUS[724].Status := 0;
   STATUS[724].TimeStamp := 16#0000;
   STATUS[725].EXT.AlarmWarnUnAck := FALSE;
   STATUS[725].EXT.AckRequired := FALSE;
   STATUS[725].EXT.Maintanence := FALSE;
   STATUS[725].EXT.Operation := FALSE;
   STATUS[725].EXT.Forced := FALSE;
   STATUS[725].EXT.BIT29 := FALSE;
   STATUS[725].EXT.BIT30 := FALSE;
   STATUS[725].EXT.BIT31 := FALSE;
   STATUS[725].EXT.ModeBit1 := FALSE;
   STATUS[725].EXT.ModeBit2 := FALSE;
   STATUS[725].EXT.ModeBit3 := FALSE;
   STATUS[725].EXT.BIT19 := FALSE;
   STATUS[725].EXT.BIT20 := FALSE;
   STATUS[725].EXT.AlarmSuppressed := FALSE;
   STATUS[725].EXT.AlarmPresent := FALSE;
   STATUS[725].EXT.AlarmFailUnAck := FALSE;
   STATUS[725].Status := 0;
   STATUS[725].TimeStamp := 16#0000;
   STATUS[726].EXT.AlarmWarnUnAck := FALSE;
   STATUS[726].EXT.AckRequired := FALSE;
   STATUS[726].EXT.Maintanence := FALSE;
   STATUS[726].EXT.Operation := FALSE;
   STATUS[726].EXT.Forced := FALSE;
   STATUS[726].EXT.BIT29 := FALSE;
   STATUS[726].EXT.BIT30 := FALSE;
   STATUS[726].EXT.BIT31 := FALSE;
   STATUS[726].EXT.ModeBit1 := FALSE;
   STATUS[726].EXT.ModeBit2 := FALSE;
   STATUS[726].EXT.ModeBit3 := FALSE;
   STATUS[726].EXT.BIT19 := FALSE;
   STATUS[726].EXT.BIT20 := FALSE;
   STATUS[726].EXT.AlarmSuppressed := FALSE;
   STATUS[726].EXT.AlarmPresent := FALSE;
   STATUS[726].EXT.AlarmFailUnAck := FALSE;
   STATUS[726].Status := 0;
   STATUS[726].TimeStamp := 16#0000;
   STATUS[727].EXT.AlarmWarnUnAck := FALSE;
   STATUS[727].EXT.AckRequired := FALSE;
   STATUS[727].EXT.Maintanence := FALSE;
   STATUS[727].EXT.Operation := FALSE;
   STATUS[727].EXT.Forced := FALSE;
   STATUS[727].EXT.BIT29 := FALSE;
   STATUS[727].EXT.BIT30 := FALSE;
   STATUS[727].EXT.BIT31 := FALSE;
   STATUS[727].EXT.ModeBit1 := FALSE;
   STATUS[727].EXT.ModeBit2 := FALSE;
   STATUS[727].EXT.ModeBit3 := FALSE;
   STATUS[727].EXT.BIT19 := FALSE;
   STATUS[727].EXT.BIT20 := FALSE;
   STATUS[727].EXT.AlarmSuppressed := FALSE;
   STATUS[727].EXT.AlarmPresent := FALSE;
   STATUS[727].EXT.AlarmFailUnAck := FALSE;
   STATUS[727].Status := 0;
   STATUS[727].TimeStamp := 16#0000;
   STATUS[728].EXT.AlarmWarnUnAck := FALSE;
   STATUS[728].EXT.AckRequired := FALSE;
   STATUS[728].EXT.Maintanence := FALSE;
   STATUS[728].EXT.Operation := FALSE;
   STATUS[728].EXT.Forced := FALSE;
   STATUS[728].EXT.BIT29 := FALSE;
   STATUS[728].EXT.BIT30 := FALSE;
   STATUS[728].EXT.BIT31 := FALSE;
   STATUS[728].EXT.ModeBit1 := FALSE;
   STATUS[728].EXT.ModeBit2 := FALSE;
   STATUS[728].EXT.ModeBit3 := FALSE;
   STATUS[728].EXT.BIT19 := FALSE;
   STATUS[728].EXT.BIT20 := FALSE;
   STATUS[728].EXT.AlarmSuppressed := FALSE;
   STATUS[728].EXT.AlarmPresent := FALSE;
   STATUS[728].EXT.AlarmFailUnAck := FALSE;
   STATUS[728].Status := 0;
   STATUS[728].TimeStamp := 16#0000;
   STATUS[729].EXT.AlarmWarnUnAck := FALSE;
   STATUS[729].EXT.AckRequired := FALSE;
   STATUS[729].EXT.Maintanence := FALSE;
   STATUS[729].EXT.Operation := FALSE;
   STATUS[729].EXT.Forced := FALSE;
   STATUS[729].EXT.BIT29 := FALSE;
   STATUS[729].EXT.BIT30 := FALSE;
   STATUS[729].EXT.BIT31 := FALSE;
   STATUS[729].EXT.ModeBit1 := FALSE;
   STATUS[729].EXT.ModeBit2 := FALSE;
   STATUS[729].EXT.ModeBit3 := FALSE;
   STATUS[729].EXT.BIT19 := FALSE;
   STATUS[729].EXT.BIT20 := FALSE;
   STATUS[729].EXT.AlarmSuppressed := FALSE;
   STATUS[729].EXT.AlarmPresent := FALSE;
   STATUS[729].EXT.AlarmFailUnAck := FALSE;
   STATUS[729].Status := 0;
   STATUS[729].TimeStamp := 16#0000;
   STATUS[730].EXT.AlarmWarnUnAck := FALSE;
   STATUS[730].EXT.AckRequired := FALSE;
   STATUS[730].EXT.Maintanence := FALSE;
   STATUS[730].EXT.Operation := FALSE;
   STATUS[730].EXT.Forced := FALSE;
   STATUS[730].EXT.BIT29 := FALSE;
   STATUS[730].EXT.BIT30 := FALSE;
   STATUS[730].EXT.BIT31 := FALSE;
   STATUS[730].EXT.ModeBit1 := FALSE;
   STATUS[730].EXT.ModeBit2 := FALSE;
   STATUS[730].EXT.ModeBit3 := FALSE;
   STATUS[730].EXT.BIT19 := FALSE;
   STATUS[730].EXT.BIT20 := FALSE;
   STATUS[730].EXT.AlarmSuppressed := FALSE;
   STATUS[730].EXT.AlarmPresent := FALSE;
   STATUS[730].EXT.AlarmFailUnAck := FALSE;
   STATUS[730].Status := 0;
   STATUS[730].TimeStamp := 16#0000;
   STATUS[731].EXT.AlarmWarnUnAck := FALSE;
   STATUS[731].EXT.AckRequired := FALSE;
   STATUS[731].EXT.Maintanence := FALSE;
   STATUS[731].EXT.Operation := FALSE;
   STATUS[731].EXT.Forced := FALSE;
   STATUS[731].EXT.BIT29 := FALSE;
   STATUS[731].EXT.BIT30 := FALSE;
   STATUS[731].EXT.BIT31 := FALSE;
   STATUS[731].EXT.ModeBit1 := FALSE;
   STATUS[731].EXT.ModeBit2 := FALSE;
   STATUS[731].EXT.ModeBit3 := FALSE;
   STATUS[731].EXT.BIT19 := FALSE;
   STATUS[731].EXT.BIT20 := FALSE;
   STATUS[731].EXT.AlarmSuppressed := FALSE;
   STATUS[731].EXT.AlarmPresent := FALSE;
   STATUS[731].EXT.AlarmFailUnAck := FALSE;
   STATUS[731].Status := 0;
   STATUS[731].TimeStamp := 16#0000;
   STATUS[732].EXT.AlarmWarnUnAck := FALSE;
   STATUS[732].EXT.AckRequired := FALSE;
   STATUS[732].EXT.Maintanence := FALSE;
   STATUS[732].EXT.Operation := FALSE;
   STATUS[732].EXT.Forced := FALSE;
   STATUS[732].EXT.BIT29 := FALSE;
   STATUS[732].EXT.BIT30 := FALSE;
   STATUS[732].EXT.BIT31 := FALSE;
   STATUS[732].EXT.ModeBit1 := FALSE;
   STATUS[732].EXT.ModeBit2 := FALSE;
   STATUS[732].EXT.ModeBit3 := FALSE;
   STATUS[732].EXT.BIT19 := FALSE;
   STATUS[732].EXT.BIT20 := FALSE;
   STATUS[732].EXT.AlarmSuppressed := FALSE;
   STATUS[732].EXT.AlarmPresent := FALSE;
   STATUS[732].EXT.AlarmFailUnAck := FALSE;
   STATUS[732].Status := 0;
   STATUS[732].TimeStamp := 16#0000;
   STATUS[733].EXT.AlarmWarnUnAck := FALSE;
   STATUS[733].EXT.AckRequired := FALSE;
   STATUS[733].EXT.Maintanence := FALSE;
   STATUS[733].EXT.Operation := FALSE;
   STATUS[733].EXT.Forced := FALSE;
   STATUS[733].EXT.BIT29 := FALSE;
   STATUS[733].EXT.BIT30 := FALSE;
   STATUS[733].EXT.BIT31 := FALSE;
   STATUS[733].EXT.ModeBit1 := FALSE;
   STATUS[733].EXT.ModeBit2 := FALSE;
   STATUS[733].EXT.ModeBit3 := FALSE;
   STATUS[733].EXT.BIT19 := FALSE;
   STATUS[733].EXT.BIT20 := FALSE;
   STATUS[733].EXT.AlarmSuppressed := FALSE;
   STATUS[733].EXT.AlarmPresent := FALSE;
   STATUS[733].EXT.AlarmFailUnAck := FALSE;
   STATUS[733].Status := 0;
   STATUS[733].TimeStamp := 16#0000;
   STATUS[734].EXT.AlarmWarnUnAck := FALSE;
   STATUS[734].EXT.AckRequired := FALSE;
   STATUS[734].EXT.Maintanence := FALSE;
   STATUS[734].EXT.Operation := FALSE;
   STATUS[734].EXT.Forced := FALSE;
   STATUS[734].EXT.BIT29 := FALSE;
   STATUS[734].EXT.BIT30 := FALSE;
   STATUS[734].EXT.BIT31 := FALSE;
   STATUS[734].EXT.ModeBit1 := FALSE;
   STATUS[734].EXT.ModeBit2 := FALSE;
   STATUS[734].EXT.ModeBit3 := FALSE;
   STATUS[734].EXT.BIT19 := FALSE;
   STATUS[734].EXT.BIT20 := FALSE;
   STATUS[734].EXT.AlarmSuppressed := FALSE;
   STATUS[734].EXT.AlarmPresent := FALSE;
   STATUS[734].EXT.AlarmFailUnAck := FALSE;
   STATUS[734].Status := 0;
   STATUS[734].TimeStamp := 16#0000;
   STATUS[735].EXT.AlarmWarnUnAck := FALSE;
   STATUS[735].EXT.AckRequired := FALSE;
   STATUS[735].EXT.Maintanence := FALSE;
   STATUS[735].EXT.Operation := FALSE;
   STATUS[735].EXT.Forced := FALSE;
   STATUS[735].EXT.BIT29 := FALSE;
   STATUS[735].EXT.BIT30 := FALSE;
   STATUS[735].EXT.BIT31 := FALSE;
   STATUS[735].EXT.ModeBit1 := FALSE;
   STATUS[735].EXT.ModeBit2 := FALSE;
   STATUS[735].EXT.ModeBit3 := FALSE;
   STATUS[735].EXT.BIT19 := FALSE;
   STATUS[735].EXT.BIT20 := FALSE;
   STATUS[735].EXT.AlarmSuppressed := FALSE;
   STATUS[735].EXT.AlarmPresent := FALSE;
   STATUS[735].EXT.AlarmFailUnAck := FALSE;
   STATUS[735].Status := 0;
   STATUS[735].TimeStamp := 16#0000;
   STATUS[736].EXT.AlarmWarnUnAck := FALSE;
   STATUS[736].EXT.AckRequired := FALSE;
   STATUS[736].EXT.Maintanence := FALSE;
   STATUS[736].EXT.Operation := FALSE;
   STATUS[736].EXT.Forced := FALSE;
   STATUS[736].EXT.BIT29 := FALSE;
   STATUS[736].EXT.BIT30 := FALSE;
   STATUS[736].EXT.BIT31 := FALSE;
   STATUS[736].EXT.ModeBit1 := FALSE;
   STATUS[736].EXT.ModeBit2 := FALSE;
   STATUS[736].EXT.ModeBit3 := FALSE;
   STATUS[736].EXT.BIT19 := FALSE;
   STATUS[736].EXT.BIT20 := FALSE;
   STATUS[736].EXT.AlarmSuppressed := FALSE;
   STATUS[736].EXT.AlarmPresent := FALSE;
   STATUS[736].EXT.AlarmFailUnAck := FALSE;
   STATUS[736].Status := 0;
   STATUS[736].TimeStamp := 16#0000;
   STATUS[737].EXT.AlarmWarnUnAck := FALSE;
   STATUS[737].EXT.AckRequired := FALSE;
   STATUS[737].EXT.Maintanence := FALSE;
   STATUS[737].EXT.Operation := FALSE;
   STATUS[737].EXT.Forced := FALSE;
   STATUS[737].EXT.BIT29 := FALSE;
   STATUS[737].EXT.BIT30 := FALSE;
   STATUS[737].EXT.BIT31 := FALSE;
   STATUS[737].EXT.ModeBit1 := FALSE;
   STATUS[737].EXT.ModeBit2 := FALSE;
   STATUS[737].EXT.ModeBit3 := FALSE;
   STATUS[737].EXT.BIT19 := FALSE;
   STATUS[737].EXT.BIT20 := FALSE;
   STATUS[737].EXT.AlarmSuppressed := FALSE;
   STATUS[737].EXT.AlarmPresent := FALSE;
   STATUS[737].EXT.AlarmFailUnAck := FALSE;
   STATUS[737].Status := 0;
   STATUS[737].TimeStamp := 16#0000;
   STATUS[738].EXT.AlarmWarnUnAck := FALSE;
   STATUS[738].EXT.AckRequired := FALSE;
   STATUS[738].EXT.Maintanence := FALSE;
   STATUS[738].EXT.Operation := FALSE;
   STATUS[738].EXT.Forced := FALSE;
   STATUS[738].EXT.BIT29 := FALSE;
   STATUS[738].EXT.BIT30 := FALSE;
   STATUS[738].EXT.BIT31 := FALSE;
   STATUS[738].EXT.ModeBit1 := FALSE;
   STATUS[738].EXT.ModeBit2 := FALSE;
   STATUS[738].EXT.ModeBit3 := FALSE;
   STATUS[738].EXT.BIT19 := FALSE;
   STATUS[738].EXT.BIT20 := FALSE;
   STATUS[738].EXT.AlarmSuppressed := FALSE;
   STATUS[738].EXT.AlarmPresent := FALSE;
   STATUS[738].EXT.AlarmFailUnAck := FALSE;
   STATUS[738].Status := 0;
   STATUS[738].TimeStamp := 16#0000;
   STATUS[739].EXT.AlarmWarnUnAck := FALSE;
   STATUS[739].EXT.AckRequired := FALSE;
   STATUS[739].EXT.Maintanence := FALSE;
   STATUS[739].EXT.Operation := FALSE;
   STATUS[739].EXT.Forced := FALSE;
   STATUS[739].EXT.BIT29 := FALSE;
   STATUS[739].EXT.BIT30 := FALSE;
   STATUS[739].EXT.BIT31 := FALSE;
   STATUS[739].EXT.ModeBit1 := FALSE;
   STATUS[739].EXT.ModeBit2 := FALSE;
   STATUS[739].EXT.ModeBit3 := FALSE;
   STATUS[739].EXT.BIT19 := FALSE;
   STATUS[739].EXT.BIT20 := FALSE;
   STATUS[739].EXT.AlarmSuppressed := FALSE;
   STATUS[739].EXT.AlarmPresent := FALSE;
   STATUS[739].EXT.AlarmFailUnAck := FALSE;
   STATUS[739].Status := 0;
   STATUS[739].TimeStamp := 16#0000;
   STATUS[740].EXT.AlarmWarnUnAck := FALSE;
   STATUS[740].EXT.AckRequired := FALSE;
   STATUS[740].EXT.Maintanence := FALSE;
   STATUS[740].EXT.Operation := FALSE;
   STATUS[740].EXT.Forced := FALSE;
   STATUS[740].EXT.BIT29 := FALSE;
   STATUS[740].EXT.BIT30 := FALSE;
   STATUS[740].EXT.BIT31 := FALSE;
   STATUS[740].EXT.ModeBit1 := FALSE;
   STATUS[740].EXT.ModeBit2 := FALSE;
   STATUS[740].EXT.ModeBit3 := FALSE;
   STATUS[740].EXT.BIT19 := FALSE;
   STATUS[740].EXT.BIT20 := FALSE;
   STATUS[740].EXT.AlarmSuppressed := FALSE;
   STATUS[740].EXT.AlarmPresent := FALSE;
   STATUS[740].EXT.AlarmFailUnAck := FALSE;
   STATUS[740].Status := 0;
   STATUS[740].TimeStamp := 16#0000;
   STATUS[741].EXT.AlarmWarnUnAck := FALSE;
   STATUS[741].EXT.AckRequired := FALSE;
   STATUS[741].EXT.Maintanence := FALSE;
   STATUS[741].EXT.Operation := FALSE;
   STATUS[741].EXT.Forced := FALSE;
   STATUS[741].EXT.BIT29 := FALSE;
   STATUS[741].EXT.BIT30 := FALSE;
   STATUS[741].EXT.BIT31 := FALSE;
   STATUS[741].EXT.ModeBit1 := FALSE;
   STATUS[741].EXT.ModeBit2 := FALSE;
   STATUS[741].EXT.ModeBit3 := FALSE;
   STATUS[741].EXT.BIT19 := FALSE;
   STATUS[741].EXT.BIT20 := FALSE;
   STATUS[741].EXT.AlarmSuppressed := FALSE;
   STATUS[741].EXT.AlarmPresent := FALSE;
   STATUS[741].EXT.AlarmFailUnAck := FALSE;
   STATUS[741].Status := 0;
   STATUS[741].TimeStamp := 16#0000;
   STATUS[742].EXT.AlarmWarnUnAck := FALSE;
   STATUS[742].EXT.AckRequired := FALSE;
   STATUS[742].EXT.Maintanence := FALSE;
   STATUS[742].EXT.Operation := FALSE;
   STATUS[742].EXT.Forced := FALSE;
   STATUS[742].EXT.BIT29 := FALSE;
   STATUS[742].EXT.BIT30 := FALSE;
   STATUS[742].EXT.BIT31 := FALSE;
   STATUS[742].EXT.ModeBit1 := FALSE;
   STATUS[742].EXT.ModeBit2 := FALSE;
   STATUS[742].EXT.ModeBit3 := FALSE;
   STATUS[742].EXT.BIT19 := FALSE;
   STATUS[742].EXT.BIT20 := FALSE;
   STATUS[742].EXT.AlarmSuppressed := FALSE;
   STATUS[742].EXT.AlarmPresent := FALSE;
   STATUS[742].EXT.AlarmFailUnAck := FALSE;
   STATUS[742].Status := 0;
   STATUS[742].TimeStamp := 16#0000;
   STATUS[743].EXT.AlarmWarnUnAck := FALSE;
   STATUS[743].EXT.AckRequired := FALSE;
   STATUS[743].EXT.Maintanence := FALSE;
   STATUS[743].EXT.Operation := FALSE;
   STATUS[743].EXT.Forced := FALSE;
   STATUS[743].EXT.BIT29 := FALSE;
   STATUS[743].EXT.BIT30 := FALSE;
   STATUS[743].EXT.BIT31 := FALSE;
   STATUS[743].EXT.ModeBit1 := FALSE;
   STATUS[743].EXT.ModeBit2 := FALSE;
   STATUS[743].EXT.ModeBit3 := FALSE;
   STATUS[743].EXT.BIT19 := FALSE;
   STATUS[743].EXT.BIT20 := FALSE;
   STATUS[743].EXT.AlarmSuppressed := FALSE;
   STATUS[743].EXT.AlarmPresent := FALSE;
   STATUS[743].EXT.AlarmFailUnAck := FALSE;
   STATUS[743].Status := 0;
   STATUS[743].TimeStamp := 16#0000;
   STATUS[744].EXT.AlarmWarnUnAck := FALSE;
   STATUS[744].EXT.AckRequired := FALSE;
   STATUS[744].EXT.Maintanence := FALSE;
   STATUS[744].EXT.Operation := FALSE;
   STATUS[744].EXT.Forced := FALSE;
   STATUS[744].EXT.BIT29 := FALSE;
   STATUS[744].EXT.BIT30 := FALSE;
   STATUS[744].EXT.BIT31 := FALSE;
   STATUS[744].EXT.ModeBit1 := FALSE;
   STATUS[744].EXT.ModeBit2 := FALSE;
   STATUS[744].EXT.ModeBit3 := FALSE;
   STATUS[744].EXT.BIT19 := FALSE;
   STATUS[744].EXT.BIT20 := FALSE;
   STATUS[744].EXT.AlarmSuppressed := FALSE;
   STATUS[744].EXT.AlarmPresent := FALSE;
   STATUS[744].EXT.AlarmFailUnAck := FALSE;
   STATUS[744].Status := 0;
   STATUS[744].TimeStamp := 16#0000;
   STATUS[745].EXT.AlarmWarnUnAck := FALSE;
   STATUS[745].EXT.AckRequired := FALSE;
   STATUS[745].EXT.Maintanence := FALSE;
   STATUS[745].EXT.Operation := FALSE;
   STATUS[745].EXT.Forced := FALSE;
   STATUS[745].EXT.BIT29 := FALSE;
   STATUS[745].EXT.BIT30 := FALSE;
   STATUS[745].EXT.BIT31 := FALSE;
   STATUS[745].EXT.ModeBit1 := FALSE;
   STATUS[745].EXT.ModeBit2 := FALSE;
   STATUS[745].EXT.ModeBit3 := FALSE;
   STATUS[745].EXT.BIT19 := FALSE;
   STATUS[745].EXT.BIT20 := FALSE;
   STATUS[745].EXT.AlarmSuppressed := FALSE;
   STATUS[745].EXT.AlarmPresent := FALSE;
   STATUS[745].EXT.AlarmFailUnAck := FALSE;
   STATUS[745].Status := 0;
   STATUS[745].TimeStamp := 16#0000;
   STATUS[746].EXT.AlarmWarnUnAck := FALSE;
   STATUS[746].EXT.AckRequired := FALSE;
   STATUS[746].EXT.Maintanence := FALSE;
   STATUS[746].EXT.Operation := FALSE;
   STATUS[746].EXT.Forced := FALSE;
   STATUS[746].EXT.BIT29 := FALSE;
   STATUS[746].EXT.BIT30 := FALSE;
   STATUS[746].EXT.BIT31 := FALSE;
   STATUS[746].EXT.ModeBit1 := FALSE;
   STATUS[746].EXT.ModeBit2 := FALSE;
   STATUS[746].EXT.ModeBit3 := FALSE;
   STATUS[746].EXT.BIT19 := FALSE;
   STATUS[746].EXT.BIT20 := FALSE;
   STATUS[746].EXT.AlarmSuppressed := FALSE;
   STATUS[746].EXT.AlarmPresent := FALSE;
   STATUS[746].EXT.AlarmFailUnAck := FALSE;
   STATUS[746].Status := 0;
   STATUS[746].TimeStamp := 16#0000;
   STATUS[747].EXT.AlarmWarnUnAck := FALSE;
   STATUS[747].EXT.AckRequired := FALSE;
   STATUS[747].EXT.Maintanence := FALSE;
   STATUS[747].EXT.Operation := FALSE;
   STATUS[747].EXT.Forced := FALSE;
   STATUS[747].EXT.BIT29 := FALSE;
   STATUS[747].EXT.BIT30 := FALSE;
   STATUS[747].EXT.BIT31 := FALSE;
   STATUS[747].EXT.ModeBit1 := FALSE;
   STATUS[747].EXT.ModeBit2 := FALSE;
   STATUS[747].EXT.ModeBit3 := FALSE;
   STATUS[747].EXT.BIT19 := FALSE;
   STATUS[747].EXT.BIT20 := FALSE;
   STATUS[747].EXT.AlarmSuppressed := FALSE;
   STATUS[747].EXT.AlarmPresent := FALSE;
   STATUS[747].EXT.AlarmFailUnAck := FALSE;
   STATUS[747].Status := 0;
   STATUS[747].TimeStamp := 16#0000;
   STATUS[748].EXT.AlarmWarnUnAck := FALSE;
   STATUS[748].EXT.AckRequired := FALSE;
   STATUS[748].EXT.Maintanence := FALSE;
   STATUS[748].EXT.Operation := FALSE;
   STATUS[748].EXT.Forced := FALSE;
   STATUS[748].EXT.BIT29 := FALSE;
   STATUS[748].EXT.BIT30 := FALSE;
   STATUS[748].EXT.BIT31 := FALSE;
   STATUS[748].EXT.ModeBit1 := FALSE;
   STATUS[748].EXT.ModeBit2 := FALSE;
   STATUS[748].EXT.ModeBit3 := FALSE;
   STATUS[748].EXT.BIT19 := FALSE;
   STATUS[748].EXT.BIT20 := FALSE;
   STATUS[748].EXT.AlarmSuppressed := FALSE;
   STATUS[748].EXT.AlarmPresent := FALSE;
   STATUS[748].EXT.AlarmFailUnAck := FALSE;
   STATUS[748].Status := 0;
   STATUS[748].TimeStamp := 16#0000;
   STATUS[749].EXT.AlarmWarnUnAck := FALSE;
   STATUS[749].EXT.AckRequired := FALSE;
   STATUS[749].EXT.Maintanence := FALSE;
   STATUS[749].EXT.Operation := FALSE;
   STATUS[749].EXT.Forced := FALSE;
   STATUS[749].EXT.BIT29 := FALSE;
   STATUS[749].EXT.BIT30 := FALSE;
   STATUS[749].EXT.BIT31 := FALSE;
   STATUS[749].EXT.ModeBit1 := FALSE;
   STATUS[749].EXT.ModeBit2 := FALSE;
   STATUS[749].EXT.ModeBit3 := FALSE;
   STATUS[749].EXT.BIT19 := FALSE;
   STATUS[749].EXT.BIT20 := FALSE;
   STATUS[749].EXT.AlarmSuppressed := FALSE;
   STATUS[749].EXT.AlarmPresent := FALSE;
   STATUS[749].EXT.AlarmFailUnAck := FALSE;
   STATUS[749].Status := 0;
   STATUS[749].TimeStamp := 16#0000;
   STATUS[750].EXT.AlarmWarnUnAck := FALSE;
   STATUS[750].EXT.AckRequired := FALSE;
   STATUS[750].EXT.Maintanence := FALSE;
   STATUS[750].EXT.Operation := FALSE;
   STATUS[750].EXT.Forced := FALSE;
   STATUS[750].EXT.BIT29 := FALSE;
   STATUS[750].EXT.BIT30 := FALSE;
   STATUS[750].EXT.BIT31 := FALSE;
   STATUS[750].EXT.ModeBit1 := FALSE;
   STATUS[750].EXT.ModeBit2 := FALSE;
   STATUS[750].EXT.ModeBit3 := FALSE;
   STATUS[750].EXT.BIT19 := FALSE;
   STATUS[750].EXT.BIT20 := FALSE;
   STATUS[750].EXT.AlarmSuppressed := FALSE;
   STATUS[750].EXT.AlarmPresent := FALSE;
   STATUS[750].EXT.AlarmFailUnAck := FALSE;
   STATUS[750].Status := 0;
   STATUS[750].TimeStamp := 16#0000;
   STATUS[751].EXT.AlarmWarnUnAck := FALSE;
   STATUS[751].EXT.AckRequired := FALSE;
   STATUS[751].EXT.Maintanence := FALSE;
   STATUS[751].EXT.Operation := FALSE;
   STATUS[751].EXT.Forced := FALSE;
   STATUS[751].EXT.BIT29 := FALSE;
   STATUS[751].EXT.BIT30 := FALSE;
   STATUS[751].EXT.BIT31 := FALSE;
   STATUS[751].EXT.ModeBit1 := FALSE;
   STATUS[751].EXT.ModeBit2 := FALSE;
   STATUS[751].EXT.ModeBit3 := FALSE;
   STATUS[751].EXT.BIT19 := FALSE;
   STATUS[751].EXT.BIT20 := FALSE;
   STATUS[751].EXT.AlarmSuppressed := FALSE;
   STATUS[751].EXT.AlarmPresent := FALSE;
   STATUS[751].EXT.AlarmFailUnAck := FALSE;
   STATUS[751].Status := 0;
   STATUS[751].TimeStamp := 16#0000;
   STATUS[752].EXT.AlarmWarnUnAck := FALSE;
   STATUS[752].EXT.AckRequired := FALSE;
   STATUS[752].EXT.Maintanence := FALSE;
   STATUS[752].EXT.Operation := FALSE;
   STATUS[752].EXT.Forced := FALSE;
   STATUS[752].EXT.BIT29 := FALSE;
   STATUS[752].EXT.BIT30 := FALSE;
   STATUS[752].EXT.BIT31 := FALSE;
   STATUS[752].EXT.ModeBit1 := FALSE;
   STATUS[752].EXT.ModeBit2 := FALSE;
   STATUS[752].EXT.ModeBit3 := FALSE;
   STATUS[752].EXT.BIT19 := FALSE;
   STATUS[752].EXT.BIT20 := FALSE;
   STATUS[752].EXT.AlarmSuppressed := FALSE;
   STATUS[752].EXT.AlarmPresent := FALSE;
   STATUS[752].EXT.AlarmFailUnAck := FALSE;
   STATUS[752].Status := 0;
   STATUS[752].TimeStamp := 16#0000;
   STATUS[753].EXT.AlarmWarnUnAck := FALSE;
   STATUS[753].EXT.AckRequired := FALSE;
   STATUS[753].EXT.Maintanence := FALSE;
   STATUS[753].EXT.Operation := FALSE;
   STATUS[753].EXT.Forced := FALSE;
   STATUS[753].EXT.BIT29 := FALSE;
   STATUS[753].EXT.BIT30 := FALSE;
   STATUS[753].EXT.BIT31 := FALSE;
   STATUS[753].EXT.ModeBit1 := FALSE;
   STATUS[753].EXT.ModeBit2 := FALSE;
   STATUS[753].EXT.ModeBit3 := FALSE;
   STATUS[753].EXT.BIT19 := FALSE;
   STATUS[753].EXT.BIT20 := FALSE;
   STATUS[753].EXT.AlarmSuppressed := FALSE;
   STATUS[753].EXT.AlarmPresent := FALSE;
   STATUS[753].EXT.AlarmFailUnAck := FALSE;
   STATUS[753].Status := 0;
   STATUS[753].TimeStamp := 16#0000;
   STATUS[754].EXT.AlarmWarnUnAck := FALSE;
   STATUS[754].EXT.AckRequired := FALSE;
   STATUS[754].EXT.Maintanence := FALSE;
   STATUS[754].EXT.Operation := FALSE;
   STATUS[754].EXT.Forced := FALSE;
   STATUS[754].EXT.BIT29 := FALSE;
   STATUS[754].EXT.BIT30 := FALSE;
   STATUS[754].EXT.BIT31 := FALSE;
   STATUS[754].EXT.ModeBit1 := FALSE;
   STATUS[754].EXT.ModeBit2 := FALSE;
   STATUS[754].EXT.ModeBit3 := FALSE;
   STATUS[754].EXT.BIT19 := FALSE;
   STATUS[754].EXT.BIT20 := FALSE;
   STATUS[754].EXT.AlarmSuppressed := FALSE;
   STATUS[754].EXT.AlarmPresent := FALSE;
   STATUS[754].EXT.AlarmFailUnAck := FALSE;
   STATUS[754].Status := 0;
   STATUS[754].TimeStamp := 16#0000;
   STATUS[755].EXT.AlarmWarnUnAck := FALSE;
   STATUS[755].EXT.AckRequired := FALSE;
   STATUS[755].EXT.Maintanence := FALSE;
   STATUS[755].EXT.Operation := FALSE;
   STATUS[755].EXT.Forced := FALSE;
   STATUS[755].EXT.BIT29 := FALSE;
   STATUS[755].EXT.BIT30 := FALSE;
   STATUS[755].EXT.BIT31 := FALSE;
   STATUS[755].EXT.ModeBit1 := FALSE;
   STATUS[755].EXT.ModeBit2 := FALSE;
   STATUS[755].EXT.ModeBit3 := FALSE;
   STATUS[755].EXT.BIT19 := FALSE;
   STATUS[755].EXT.BIT20 := FALSE;
   STATUS[755].EXT.AlarmSuppressed := FALSE;
   STATUS[755].EXT.AlarmPresent := FALSE;
   STATUS[755].EXT.AlarmFailUnAck := FALSE;
   STATUS[755].Status := 0;
   STATUS[755].TimeStamp := 16#0000;
   STATUS[756].EXT.AlarmWarnUnAck := FALSE;
   STATUS[756].EXT.AckRequired := FALSE;
   STATUS[756].EXT.Maintanence := FALSE;
   STATUS[756].EXT.Operation := FALSE;
   STATUS[756].EXT.Forced := FALSE;
   STATUS[756].EXT.BIT29 := FALSE;
   STATUS[756].EXT.BIT30 := FALSE;
   STATUS[756].EXT.BIT31 := FALSE;
   STATUS[756].EXT.ModeBit1 := FALSE;
   STATUS[756].EXT.ModeBit2 := FALSE;
   STATUS[756].EXT.ModeBit3 := FALSE;
   STATUS[756].EXT.BIT19 := FALSE;
   STATUS[756].EXT.BIT20 := FALSE;
   STATUS[756].EXT.AlarmSuppressed := FALSE;
   STATUS[756].EXT.AlarmPresent := FALSE;
   STATUS[756].EXT.AlarmFailUnAck := FALSE;
   STATUS[756].Status := 0;
   STATUS[756].TimeStamp := 16#0000;
   STATUS[757].EXT.AlarmWarnUnAck := FALSE;
   STATUS[757].EXT.AckRequired := FALSE;
   STATUS[757].EXT.Maintanence := FALSE;
   STATUS[757].EXT.Operation := FALSE;
   STATUS[757].EXT.Forced := FALSE;
   STATUS[757].EXT.BIT29 := FALSE;
   STATUS[757].EXT.BIT30 := FALSE;
   STATUS[757].EXT.BIT31 := FALSE;
   STATUS[757].EXT.ModeBit1 := FALSE;
   STATUS[757].EXT.ModeBit2 := FALSE;
   STATUS[757].EXT.ModeBit3 := FALSE;
   STATUS[757].EXT.BIT19 := FALSE;
   STATUS[757].EXT.BIT20 := FALSE;
   STATUS[757].EXT.AlarmSuppressed := FALSE;
   STATUS[757].EXT.AlarmPresent := FALSE;
   STATUS[757].EXT.AlarmFailUnAck := FALSE;
   STATUS[757].Status := 0;
   STATUS[757].TimeStamp := 16#0000;
   STATUS[758].EXT.AlarmWarnUnAck := FALSE;
   STATUS[758].EXT.AckRequired := FALSE;
   STATUS[758].EXT.Maintanence := FALSE;
   STATUS[758].EXT.Operation := FALSE;
   STATUS[758].EXT.Forced := FALSE;
   STATUS[758].EXT.BIT29 := FALSE;
   STATUS[758].EXT.BIT30 := FALSE;
   STATUS[758].EXT.BIT31 := FALSE;
   STATUS[758].EXT.ModeBit1 := FALSE;
   STATUS[758].EXT.ModeBit2 := FALSE;
   STATUS[758].EXT.ModeBit3 := FALSE;
   STATUS[758].EXT.BIT19 := FALSE;
   STATUS[758].EXT.BIT20 := FALSE;
   STATUS[758].EXT.AlarmSuppressed := FALSE;
   STATUS[758].EXT.AlarmPresent := FALSE;
   STATUS[758].EXT.AlarmFailUnAck := FALSE;
   STATUS[758].Status := 0;
   STATUS[758].TimeStamp := 16#0000;
   STATUS[759].EXT.AlarmWarnUnAck := FALSE;
   STATUS[759].EXT.AckRequired := FALSE;
   STATUS[759].EXT.Maintanence := FALSE;
   STATUS[759].EXT.Operation := FALSE;
   STATUS[759].EXT.Forced := FALSE;
   STATUS[759].EXT.BIT29 := FALSE;
   STATUS[759].EXT.BIT30 := FALSE;
   STATUS[759].EXT.BIT31 := FALSE;
   STATUS[759].EXT.ModeBit1 := FALSE;
   STATUS[759].EXT.ModeBit2 := FALSE;
   STATUS[759].EXT.ModeBit3 := FALSE;
   STATUS[759].EXT.BIT19 := FALSE;
   STATUS[759].EXT.BIT20 := FALSE;
   STATUS[759].EXT.AlarmSuppressed := FALSE;
   STATUS[759].EXT.AlarmPresent := FALSE;
   STATUS[759].EXT.AlarmFailUnAck := FALSE;
   STATUS[759].Status := 0;
   STATUS[759].TimeStamp := 16#0000;
   STATUS[760].EXT.AlarmWarnUnAck := FALSE;
   STATUS[760].EXT.AckRequired := FALSE;
   STATUS[760].EXT.Maintanence := FALSE;
   STATUS[760].EXT.Operation := FALSE;
   STATUS[760].EXT.Forced := FALSE;
   STATUS[760].EXT.BIT29 := FALSE;
   STATUS[760].EXT.BIT30 := FALSE;
   STATUS[760].EXT.BIT31 := FALSE;
   STATUS[760].EXT.ModeBit1 := FALSE;
   STATUS[760].EXT.ModeBit2 := FALSE;
   STATUS[760].EXT.ModeBit3 := FALSE;
   STATUS[760].EXT.BIT19 := FALSE;
   STATUS[760].EXT.BIT20 := FALSE;
   STATUS[760].EXT.AlarmSuppressed := FALSE;
   STATUS[760].EXT.AlarmPresent := FALSE;
   STATUS[760].EXT.AlarmFailUnAck := FALSE;
   STATUS[760].Status := 0;
   STATUS[760].TimeStamp := 16#0000;
   STATUS[761].EXT.AlarmWarnUnAck := FALSE;
   STATUS[761].EXT.AckRequired := FALSE;
   STATUS[761].EXT.Maintanence := FALSE;
   STATUS[761].EXT.Operation := FALSE;
   STATUS[761].EXT.Forced := FALSE;
   STATUS[761].EXT.BIT29 := FALSE;
   STATUS[761].EXT.BIT30 := FALSE;
   STATUS[761].EXT.BIT31 := FALSE;
   STATUS[761].EXT.ModeBit1 := FALSE;
   STATUS[761].EXT.ModeBit2 := FALSE;
   STATUS[761].EXT.ModeBit3 := FALSE;
   STATUS[761].EXT.BIT19 := FALSE;
   STATUS[761].EXT.BIT20 := FALSE;
   STATUS[761].EXT.AlarmSuppressed := FALSE;
   STATUS[761].EXT.AlarmPresent := FALSE;
   STATUS[761].EXT.AlarmFailUnAck := FALSE;
   STATUS[761].Status := 0;
   STATUS[761].TimeStamp := 16#0000;
   STATUS[762].EXT.AlarmWarnUnAck := FALSE;
   STATUS[762].EXT.AckRequired := FALSE;
   STATUS[762].EXT.Maintanence := FALSE;
   STATUS[762].EXT.Operation := FALSE;
   STATUS[762].EXT.Forced := FALSE;
   STATUS[762].EXT.BIT29 := FALSE;
   STATUS[762].EXT.BIT30 := FALSE;
   STATUS[762].EXT.BIT31 := FALSE;
   STATUS[762].EXT.ModeBit1 := FALSE;
   STATUS[762].EXT.ModeBit2 := FALSE;
   STATUS[762].EXT.ModeBit3 := FALSE;
   STATUS[762].EXT.BIT19 := FALSE;
   STATUS[762].EXT.BIT20 := FALSE;
   STATUS[762].EXT.AlarmSuppressed := FALSE;
   STATUS[762].EXT.AlarmPresent := FALSE;
   STATUS[762].EXT.AlarmFailUnAck := FALSE;
   STATUS[762].Status := 0;
   STATUS[762].TimeStamp := 16#0000;
   STATUS[763].EXT.AlarmWarnUnAck := FALSE;
   STATUS[763].EXT.AckRequired := FALSE;
   STATUS[763].EXT.Maintanence := FALSE;
   STATUS[763].EXT.Operation := FALSE;
   STATUS[763].EXT.Forced := FALSE;
   STATUS[763].EXT.BIT29 := FALSE;
   STATUS[763].EXT.BIT30 := FALSE;
   STATUS[763].EXT.BIT31 := FALSE;
   STATUS[763].EXT.ModeBit1 := FALSE;
   STATUS[763].EXT.ModeBit2 := FALSE;
   STATUS[763].EXT.ModeBit3 := FALSE;
   STATUS[763].EXT.BIT19 := FALSE;
   STATUS[763].EXT.BIT20 := FALSE;
   STATUS[763].EXT.AlarmSuppressed := FALSE;
   STATUS[763].EXT.AlarmPresent := FALSE;
   STATUS[763].EXT.AlarmFailUnAck := FALSE;
   STATUS[763].Status := 0;
   STATUS[763].TimeStamp := 16#0000;
   STATUS[764].EXT.AlarmWarnUnAck := FALSE;
   STATUS[764].EXT.AckRequired := FALSE;
   STATUS[764].EXT.Maintanence := FALSE;
   STATUS[764].EXT.Operation := FALSE;
   STATUS[764].EXT.Forced := FALSE;
   STATUS[764].EXT.BIT29 := FALSE;
   STATUS[764].EXT.BIT30 := FALSE;
   STATUS[764].EXT.BIT31 := FALSE;
   STATUS[764].EXT.ModeBit1 := FALSE;
   STATUS[764].EXT.ModeBit2 := FALSE;
   STATUS[764].EXT.ModeBit3 := FALSE;
   STATUS[764].EXT.BIT19 := FALSE;
   STATUS[764].EXT.BIT20 := FALSE;
   STATUS[764].EXT.AlarmSuppressed := FALSE;
   STATUS[764].EXT.AlarmPresent := FALSE;
   STATUS[764].EXT.AlarmFailUnAck := FALSE;
   STATUS[764].Status := 0;
   STATUS[764].TimeStamp := 16#0000;
   STATUS[765].EXT.AlarmWarnUnAck := FALSE;
   STATUS[765].EXT.AckRequired := FALSE;
   STATUS[765].EXT.Maintanence := FALSE;
   STATUS[765].EXT.Operation := FALSE;
   STATUS[765].EXT.Forced := FALSE;
   STATUS[765].EXT.BIT29 := FALSE;
   STATUS[765].EXT.BIT30 := FALSE;
   STATUS[765].EXT.BIT31 := FALSE;
   STATUS[765].EXT.ModeBit1 := FALSE;
   STATUS[765].EXT.ModeBit2 := FALSE;
   STATUS[765].EXT.ModeBit3 := FALSE;
   STATUS[765].EXT.BIT19 := FALSE;
   STATUS[765].EXT.BIT20 := FALSE;
   STATUS[765].EXT.AlarmSuppressed := FALSE;
   STATUS[765].EXT.AlarmPresent := FALSE;
   STATUS[765].EXT.AlarmFailUnAck := FALSE;
   STATUS[765].Status := 0;
   STATUS[765].TimeStamp := 16#0000;
   STATUS[766].EXT.AlarmWarnUnAck := FALSE;
   STATUS[766].EXT.AckRequired := FALSE;
   STATUS[766].EXT.Maintanence := FALSE;
   STATUS[766].EXT.Operation := FALSE;
   STATUS[766].EXT.Forced := FALSE;
   STATUS[766].EXT.BIT29 := FALSE;
   STATUS[766].EXT.BIT30 := FALSE;
   STATUS[766].EXT.BIT31 := FALSE;
   STATUS[766].EXT.ModeBit1 := FALSE;
   STATUS[766].EXT.ModeBit2 := FALSE;
   STATUS[766].EXT.ModeBit3 := FALSE;
   STATUS[766].EXT.BIT19 := FALSE;
   STATUS[766].EXT.BIT20 := FALSE;
   STATUS[766].EXT.AlarmSuppressed := FALSE;
   STATUS[766].EXT.AlarmPresent := FALSE;
   STATUS[766].EXT.AlarmFailUnAck := FALSE;
   STATUS[766].Status := 0;
   STATUS[766].TimeStamp := 16#0000;
   STATUS[767].EXT.AlarmWarnUnAck := FALSE;
   STATUS[767].EXT.AckRequired := FALSE;
   STATUS[767].EXT.Maintanence := FALSE;
   STATUS[767].EXT.Operation := FALSE;
   STATUS[767].EXT.Forced := FALSE;
   STATUS[767].EXT.BIT29 := FALSE;
   STATUS[767].EXT.BIT30 := FALSE;
   STATUS[767].EXT.BIT31 := FALSE;
   STATUS[767].EXT.ModeBit1 := FALSE;
   STATUS[767].EXT.ModeBit2 := FALSE;
   STATUS[767].EXT.ModeBit3 := FALSE;
   STATUS[767].EXT.BIT19 := FALSE;
   STATUS[767].EXT.BIT20 := FALSE;
   STATUS[767].EXT.AlarmSuppressed := FALSE;
   STATUS[767].EXT.AlarmPresent := FALSE;
   STATUS[767].EXT.AlarmFailUnAck := FALSE;
   STATUS[767].Status := 0;
   STATUS[767].TimeStamp := 16#0000;
   STATUS[768].EXT.AlarmWarnUnAck := FALSE;
   STATUS[768].EXT.AckRequired := FALSE;
   STATUS[768].EXT.Maintanence := FALSE;
   STATUS[768].EXT.Operation := FALSE;
   STATUS[768].EXT.Forced := FALSE;
   STATUS[768].EXT.BIT29 := FALSE;
   STATUS[768].EXT.BIT30 := FALSE;
   STATUS[768].EXT.BIT31 := FALSE;
   STATUS[768].EXT.ModeBit1 := FALSE;
   STATUS[768].EXT.ModeBit2 := FALSE;
   STATUS[768].EXT.ModeBit3 := FALSE;
   STATUS[768].EXT.BIT19 := FALSE;
   STATUS[768].EXT.BIT20 := FALSE;
   STATUS[768].EXT.AlarmSuppressed := FALSE;
   STATUS[768].EXT.AlarmPresent := FALSE;
   STATUS[768].EXT.AlarmFailUnAck := FALSE;
   STATUS[768].Status := 0;
   STATUS[768].TimeStamp := 16#0000;
   STATUS[769].EXT.AlarmWarnUnAck := FALSE;
   STATUS[769].EXT.AckRequired := FALSE;
   STATUS[769].EXT.Maintanence := FALSE;
   STATUS[769].EXT.Operation := FALSE;
   STATUS[769].EXT.Forced := FALSE;
   STATUS[769].EXT.BIT29 := FALSE;
   STATUS[769].EXT.BIT30 := FALSE;
   STATUS[769].EXT.BIT31 := FALSE;
   STATUS[769].EXT.ModeBit1 := FALSE;
   STATUS[769].EXT.ModeBit2 := FALSE;
   STATUS[769].EXT.ModeBit3 := FALSE;
   STATUS[769].EXT.BIT19 := FALSE;
   STATUS[769].EXT.BIT20 := FALSE;
   STATUS[769].EXT.AlarmSuppressed := FALSE;
   STATUS[769].EXT.AlarmPresent := FALSE;
   STATUS[769].EXT.AlarmFailUnAck := FALSE;
   STATUS[769].Status := 0;
   STATUS[769].TimeStamp := 16#0000;
   STATUS[770].EXT.AlarmWarnUnAck := FALSE;
   STATUS[770].EXT.AckRequired := FALSE;
   STATUS[770].EXT.Maintanence := FALSE;
   STATUS[770].EXT.Operation := FALSE;
   STATUS[770].EXT.Forced := FALSE;
   STATUS[770].EXT.BIT29 := FALSE;
   STATUS[770].EXT.BIT30 := FALSE;
   STATUS[770].EXT.BIT31 := FALSE;
   STATUS[770].EXT.ModeBit1 := FALSE;
   STATUS[770].EXT.ModeBit2 := FALSE;
   STATUS[770].EXT.ModeBit3 := FALSE;
   STATUS[770].EXT.BIT19 := FALSE;
   STATUS[770].EXT.BIT20 := FALSE;
   STATUS[770].EXT.AlarmSuppressed := FALSE;
   STATUS[770].EXT.AlarmPresent := FALSE;
   STATUS[770].EXT.AlarmFailUnAck := FALSE;
   STATUS[770].Status := 0;
   STATUS[770].TimeStamp := 16#0000;
   STATUS[771].EXT.AlarmWarnUnAck := FALSE;
   STATUS[771].EXT.AckRequired := FALSE;
   STATUS[771].EXT.Maintanence := FALSE;
   STATUS[771].EXT.Operation := FALSE;
   STATUS[771].EXT.Forced := FALSE;
   STATUS[771].EXT.BIT29 := FALSE;
   STATUS[771].EXT.BIT30 := FALSE;
   STATUS[771].EXT.BIT31 := FALSE;
   STATUS[771].EXT.ModeBit1 := FALSE;
   STATUS[771].EXT.ModeBit2 := FALSE;
   STATUS[771].EXT.ModeBit3 := FALSE;
   STATUS[771].EXT.BIT19 := FALSE;
   STATUS[771].EXT.BIT20 := FALSE;
   STATUS[771].EXT.AlarmSuppressed := FALSE;
   STATUS[771].EXT.AlarmPresent := FALSE;
   STATUS[771].EXT.AlarmFailUnAck := FALSE;
   STATUS[771].Status := 0;
   STATUS[771].TimeStamp := 16#0000;
   STATUS[772].EXT.AlarmWarnUnAck := FALSE;
   STATUS[772].EXT.AckRequired := FALSE;
   STATUS[772].EXT.Maintanence := FALSE;
   STATUS[772].EXT.Operation := FALSE;
   STATUS[772].EXT.Forced := FALSE;
   STATUS[772].EXT.BIT29 := FALSE;
   STATUS[772].EXT.BIT30 := FALSE;
   STATUS[772].EXT.BIT31 := FALSE;
   STATUS[772].EXT.ModeBit1 := FALSE;
   STATUS[772].EXT.ModeBit2 := FALSE;
   STATUS[772].EXT.ModeBit3 := FALSE;
   STATUS[772].EXT.BIT19 := FALSE;
   STATUS[772].EXT.BIT20 := FALSE;
   STATUS[772].EXT.AlarmSuppressed := FALSE;
   STATUS[772].EXT.AlarmPresent := FALSE;
   STATUS[772].EXT.AlarmFailUnAck := FALSE;
   STATUS[772].Status := 0;
   STATUS[772].TimeStamp := 16#0000;
   STATUS[773].EXT.AlarmWarnUnAck := FALSE;
   STATUS[773].EXT.AckRequired := FALSE;
   STATUS[773].EXT.Maintanence := FALSE;
   STATUS[773].EXT.Operation := FALSE;
   STATUS[773].EXT.Forced := FALSE;
   STATUS[773].EXT.BIT29 := FALSE;
   STATUS[773].EXT.BIT30 := FALSE;
   STATUS[773].EXT.BIT31 := FALSE;
   STATUS[773].EXT.ModeBit1 := FALSE;
   STATUS[773].EXT.ModeBit2 := FALSE;
   STATUS[773].EXT.ModeBit3 := FALSE;
   STATUS[773].EXT.BIT19 := FALSE;
   STATUS[773].EXT.BIT20 := FALSE;
   STATUS[773].EXT.AlarmSuppressed := FALSE;
   STATUS[773].EXT.AlarmPresent := FALSE;
   STATUS[773].EXT.AlarmFailUnAck := FALSE;
   STATUS[773].Status := 0;
   STATUS[773].TimeStamp := 16#0000;
   STATUS[774].EXT.AlarmWarnUnAck := FALSE;
   STATUS[774].EXT.AckRequired := FALSE;
   STATUS[774].EXT.Maintanence := FALSE;
   STATUS[774].EXT.Operation := FALSE;
   STATUS[774].EXT.Forced := FALSE;
   STATUS[774].EXT.BIT29 := FALSE;
   STATUS[774].EXT.BIT30 := FALSE;
   STATUS[774].EXT.BIT31 := FALSE;
   STATUS[774].EXT.ModeBit1 := FALSE;
   STATUS[774].EXT.ModeBit2 := FALSE;
   STATUS[774].EXT.ModeBit3 := FALSE;
   STATUS[774].EXT.BIT19 := FALSE;
   STATUS[774].EXT.BIT20 := FALSE;
   STATUS[774].EXT.AlarmSuppressed := FALSE;
   STATUS[774].EXT.AlarmPresent := FALSE;
   STATUS[774].EXT.AlarmFailUnAck := FALSE;
   STATUS[774].Status := 0;
   STATUS[774].TimeStamp := 16#0000;
   STATUS[775].EXT.AlarmWarnUnAck := FALSE;
   STATUS[775].EXT.AckRequired := FALSE;
   STATUS[775].EXT.Maintanence := FALSE;
   STATUS[775].EXT.Operation := FALSE;
   STATUS[775].EXT.Forced := FALSE;
   STATUS[775].EXT.BIT29 := FALSE;
   STATUS[775].EXT.BIT30 := FALSE;
   STATUS[775].EXT.BIT31 := FALSE;
   STATUS[775].EXT.ModeBit1 := FALSE;
   STATUS[775].EXT.ModeBit2 := FALSE;
   STATUS[775].EXT.ModeBit3 := FALSE;
   STATUS[775].EXT.BIT19 := FALSE;
   STATUS[775].EXT.BIT20 := FALSE;
   STATUS[775].EXT.AlarmSuppressed := FALSE;
   STATUS[775].EXT.AlarmPresent := FALSE;
   STATUS[775].EXT.AlarmFailUnAck := FALSE;
   STATUS[775].Status := 0;
   STATUS[775].TimeStamp := 16#0000;
   STATUS[776].EXT.AlarmWarnUnAck := FALSE;
   STATUS[776].EXT.AckRequired := FALSE;
   STATUS[776].EXT.Maintanence := FALSE;
   STATUS[776].EXT.Operation := FALSE;
   STATUS[776].EXT.Forced := FALSE;
   STATUS[776].EXT.BIT29 := FALSE;
   STATUS[776].EXT.BIT30 := FALSE;
   STATUS[776].EXT.BIT31 := FALSE;
   STATUS[776].EXT.ModeBit1 := FALSE;
   STATUS[776].EXT.ModeBit2 := FALSE;
   STATUS[776].EXT.ModeBit3 := FALSE;
   STATUS[776].EXT.BIT19 := FALSE;
   STATUS[776].EXT.BIT20 := FALSE;
   STATUS[776].EXT.AlarmSuppressed := FALSE;
   STATUS[776].EXT.AlarmPresent := FALSE;
   STATUS[776].EXT.AlarmFailUnAck := FALSE;
   STATUS[776].Status := 0;
   STATUS[776].TimeStamp := 16#0000;
   STATUS[777].EXT.AlarmWarnUnAck := FALSE;
   STATUS[777].EXT.AckRequired := FALSE;
   STATUS[777].EXT.Maintanence := FALSE;
   STATUS[777].EXT.Operation := FALSE;
   STATUS[777].EXT.Forced := FALSE;
   STATUS[777].EXT.BIT29 := FALSE;
   STATUS[777].EXT.BIT30 := FALSE;
   STATUS[777].EXT.BIT31 := FALSE;
   STATUS[777].EXT.ModeBit1 := FALSE;
   STATUS[777].EXT.ModeBit2 := FALSE;
   STATUS[777].EXT.ModeBit3 := FALSE;
   STATUS[777].EXT.BIT19 := FALSE;
   STATUS[777].EXT.BIT20 := FALSE;
   STATUS[777].EXT.AlarmSuppressed := FALSE;
   STATUS[777].EXT.AlarmPresent := FALSE;
   STATUS[777].EXT.AlarmFailUnAck := FALSE;
   STATUS[777].Status := 0;
   STATUS[777].TimeStamp := 16#0000;
   STATUS[778].EXT.AlarmWarnUnAck := FALSE;
   STATUS[778].EXT.AckRequired := FALSE;
   STATUS[778].EXT.Maintanence := FALSE;
   STATUS[778].EXT.Operation := FALSE;
   STATUS[778].EXT.Forced := FALSE;
   STATUS[778].EXT.BIT29 := FALSE;
   STATUS[778].EXT.BIT30 := FALSE;
   STATUS[778].EXT.BIT31 := FALSE;
   STATUS[778].EXT.ModeBit1 := FALSE;
   STATUS[778].EXT.ModeBit2 := FALSE;
   STATUS[778].EXT.ModeBit3 := FALSE;
   STATUS[778].EXT.BIT19 := FALSE;
   STATUS[778].EXT.BIT20 := FALSE;
   STATUS[778].EXT.AlarmSuppressed := FALSE;
   STATUS[778].EXT.AlarmPresent := FALSE;
   STATUS[778].EXT.AlarmFailUnAck := FALSE;
   STATUS[778].Status := 0;
   STATUS[778].TimeStamp := 16#0000;
   STATUS[779].EXT.AlarmWarnUnAck := FALSE;
   STATUS[779].EXT.AckRequired := FALSE;
   STATUS[779].EXT.Maintanence := FALSE;
   STATUS[779].EXT.Operation := FALSE;
   STATUS[779].EXT.Forced := FALSE;
   STATUS[779].EXT.BIT29 := FALSE;
   STATUS[779].EXT.BIT30 := FALSE;
   STATUS[779].EXT.BIT31 := FALSE;
   STATUS[779].EXT.ModeBit1 := FALSE;
   STATUS[779].EXT.ModeBit2 := FALSE;
   STATUS[779].EXT.ModeBit3 := FALSE;
   STATUS[779].EXT.BIT19 := FALSE;
   STATUS[779].EXT.BIT20 := FALSE;
   STATUS[779].EXT.AlarmSuppressed := FALSE;
   STATUS[779].EXT.AlarmPresent := FALSE;
   STATUS[779].EXT.AlarmFailUnAck := FALSE;
   STATUS[779].Status := 0;
   STATUS[779].TimeStamp := 16#0000;
   STATUS[780].EXT.AlarmWarnUnAck := FALSE;
   STATUS[780].EXT.AckRequired := FALSE;
   STATUS[780].EXT.Maintanence := FALSE;
   STATUS[780].EXT.Operation := FALSE;
   STATUS[780].EXT.Forced := FALSE;
   STATUS[780].EXT.BIT29 := FALSE;
   STATUS[780].EXT.BIT30 := FALSE;
   STATUS[780].EXT.BIT31 := FALSE;
   STATUS[780].EXT.ModeBit1 := FALSE;
   STATUS[780].EXT.ModeBit2 := FALSE;
   STATUS[780].EXT.ModeBit3 := FALSE;
   STATUS[780].EXT.BIT19 := FALSE;
   STATUS[780].EXT.BIT20 := FALSE;
   STATUS[780].EXT.AlarmSuppressed := FALSE;
   STATUS[780].EXT.AlarmPresent := FALSE;
   STATUS[780].EXT.AlarmFailUnAck := FALSE;
   STATUS[780].Status := 0;
   STATUS[780].TimeStamp := 16#0000;
   STATUS[781].EXT.AlarmWarnUnAck := FALSE;
   STATUS[781].EXT.AckRequired := FALSE;
   STATUS[781].EXT.Maintanence := FALSE;
   STATUS[781].EXT.Operation := FALSE;
   STATUS[781].EXT.Forced := FALSE;
   STATUS[781].EXT.BIT29 := FALSE;
   STATUS[781].EXT.BIT30 := FALSE;
   STATUS[781].EXT.BIT31 := FALSE;
   STATUS[781].EXT.ModeBit1 := FALSE;
   STATUS[781].EXT.ModeBit2 := FALSE;
   STATUS[781].EXT.ModeBit3 := FALSE;
   STATUS[781].EXT.BIT19 := FALSE;
   STATUS[781].EXT.BIT20 := FALSE;
   STATUS[781].EXT.AlarmSuppressed := FALSE;
   STATUS[781].EXT.AlarmPresent := FALSE;
   STATUS[781].EXT.AlarmFailUnAck := FALSE;
   STATUS[781].Status := 0;
   STATUS[781].TimeStamp := 16#0000;
   STATUS[782].EXT.AlarmWarnUnAck := FALSE;
   STATUS[782].EXT.AckRequired := FALSE;
   STATUS[782].EXT.Maintanence := FALSE;
   STATUS[782].EXT.Operation := FALSE;
   STATUS[782].EXT.Forced := FALSE;
   STATUS[782].EXT.BIT29 := FALSE;
   STATUS[782].EXT.BIT30 := FALSE;
   STATUS[782].EXT.BIT31 := FALSE;
   STATUS[782].EXT.ModeBit1 := FALSE;
   STATUS[782].EXT.ModeBit2 := FALSE;
   STATUS[782].EXT.ModeBit3 := FALSE;
   STATUS[782].EXT.BIT19 := FALSE;
   STATUS[782].EXT.BIT20 := FALSE;
   STATUS[782].EXT.AlarmSuppressed := FALSE;
   STATUS[782].EXT.AlarmPresent := FALSE;
   STATUS[782].EXT.AlarmFailUnAck := FALSE;
   STATUS[782].Status := 0;
   STATUS[782].TimeStamp := 16#0000;
   STATUS[783].EXT.AlarmWarnUnAck := FALSE;
   STATUS[783].EXT.AckRequired := FALSE;
   STATUS[783].EXT.Maintanence := FALSE;
   STATUS[783].EXT.Operation := FALSE;
   STATUS[783].EXT.Forced := FALSE;
   STATUS[783].EXT.BIT29 := FALSE;
   STATUS[783].EXT.BIT30 := FALSE;
   STATUS[783].EXT.BIT31 := FALSE;
   STATUS[783].EXT.ModeBit1 := FALSE;
   STATUS[783].EXT.ModeBit2 := FALSE;
   STATUS[783].EXT.ModeBit3 := FALSE;
   STATUS[783].EXT.BIT19 := FALSE;
   STATUS[783].EXT.BIT20 := FALSE;
   STATUS[783].EXT.AlarmSuppressed := FALSE;
   STATUS[783].EXT.AlarmPresent := FALSE;
   STATUS[783].EXT.AlarmFailUnAck := FALSE;
   STATUS[783].Status := 0;
   STATUS[783].TimeStamp := 16#0000;
   STATUS[784].EXT.AlarmWarnUnAck := FALSE;
   STATUS[784].EXT.AckRequired := FALSE;
   STATUS[784].EXT.Maintanence := FALSE;
   STATUS[784].EXT.Operation := FALSE;
   STATUS[784].EXT.Forced := FALSE;
   STATUS[784].EXT.BIT29 := FALSE;
   STATUS[784].EXT.BIT30 := FALSE;
   STATUS[784].EXT.BIT31 := FALSE;
   STATUS[784].EXT.ModeBit1 := FALSE;
   STATUS[784].EXT.ModeBit2 := FALSE;
   STATUS[784].EXT.ModeBit3 := FALSE;
   STATUS[784].EXT.BIT19 := FALSE;
   STATUS[784].EXT.BIT20 := FALSE;
   STATUS[784].EXT.AlarmSuppressed := FALSE;
   STATUS[784].EXT.AlarmPresent := FALSE;
   STATUS[784].EXT.AlarmFailUnAck := FALSE;
   STATUS[784].Status := 0;
   STATUS[784].TimeStamp := 16#0000;
   STATUS[785].EXT.AlarmWarnUnAck := FALSE;
   STATUS[785].EXT.AckRequired := FALSE;
   STATUS[785].EXT.Maintanence := FALSE;
   STATUS[785].EXT.Operation := FALSE;
   STATUS[785].EXT.Forced := FALSE;
   STATUS[785].EXT.BIT29 := FALSE;
   STATUS[785].EXT.BIT30 := FALSE;
   STATUS[785].EXT.BIT31 := FALSE;
   STATUS[785].EXT.ModeBit1 := FALSE;
   STATUS[785].EXT.ModeBit2 := FALSE;
   STATUS[785].EXT.ModeBit3 := FALSE;
   STATUS[785].EXT.BIT19 := FALSE;
   STATUS[785].EXT.BIT20 := FALSE;
   STATUS[785].EXT.AlarmSuppressed := FALSE;
   STATUS[785].EXT.AlarmPresent := FALSE;
   STATUS[785].EXT.AlarmFailUnAck := FALSE;
   STATUS[785].Status := 0;
   STATUS[785].TimeStamp := 16#0000;
   STATUS[786].EXT.AlarmWarnUnAck := FALSE;
   STATUS[786].EXT.AckRequired := FALSE;
   STATUS[786].EXT.Maintanence := FALSE;
   STATUS[786].EXT.Operation := FALSE;
   STATUS[786].EXT.Forced := FALSE;
   STATUS[786].EXT.BIT29 := FALSE;
   STATUS[786].EXT.BIT30 := FALSE;
   STATUS[786].EXT.BIT31 := FALSE;
   STATUS[786].EXT.ModeBit1 := FALSE;
   STATUS[786].EXT.ModeBit2 := FALSE;
   STATUS[786].EXT.ModeBit3 := FALSE;
   STATUS[786].EXT.BIT19 := FALSE;
   STATUS[786].EXT.BIT20 := FALSE;
   STATUS[786].EXT.AlarmSuppressed := FALSE;
   STATUS[786].EXT.AlarmPresent := FALSE;
   STATUS[786].EXT.AlarmFailUnAck := FALSE;
   STATUS[786].Status := 0;
   STATUS[786].TimeStamp := 16#0000;
   STATUS[787].EXT.AlarmWarnUnAck := FALSE;
   STATUS[787].EXT.AckRequired := FALSE;
   STATUS[787].EXT.Maintanence := FALSE;
   STATUS[787].EXT.Operation := FALSE;
   STATUS[787].EXT.Forced := FALSE;
   STATUS[787].EXT.BIT29 := FALSE;
   STATUS[787].EXT.BIT30 := FALSE;
   STATUS[787].EXT.BIT31 := FALSE;
   STATUS[787].EXT.ModeBit1 := FALSE;
   STATUS[787].EXT.ModeBit2 := FALSE;
   STATUS[787].EXT.ModeBit3 := FALSE;
   STATUS[787].EXT.BIT19 := FALSE;
   STATUS[787].EXT.BIT20 := FALSE;
   STATUS[787].EXT.AlarmSuppressed := FALSE;
   STATUS[787].EXT.AlarmPresent := FALSE;
   STATUS[787].EXT.AlarmFailUnAck := FALSE;
   STATUS[787].Status := 0;
   STATUS[787].TimeStamp := 16#0000;
   STATUS[788].EXT.AlarmWarnUnAck := FALSE;
   STATUS[788].EXT.AckRequired := FALSE;
   STATUS[788].EXT.Maintanence := FALSE;
   STATUS[788].EXT.Operation := FALSE;
   STATUS[788].EXT.Forced := FALSE;
   STATUS[788].EXT.BIT29 := FALSE;
   STATUS[788].EXT.BIT30 := FALSE;
   STATUS[788].EXT.BIT31 := FALSE;
   STATUS[788].EXT.ModeBit1 := FALSE;
   STATUS[788].EXT.ModeBit2 := FALSE;
   STATUS[788].EXT.ModeBit3 := FALSE;
   STATUS[788].EXT.BIT19 := FALSE;
   STATUS[788].EXT.BIT20 := FALSE;
   STATUS[788].EXT.AlarmSuppressed := FALSE;
   STATUS[788].EXT.AlarmPresent := FALSE;
   STATUS[788].EXT.AlarmFailUnAck := FALSE;
   STATUS[788].Status := 0;
   STATUS[788].TimeStamp := 16#0000;
   STATUS[789].EXT.AlarmWarnUnAck := FALSE;
   STATUS[789].EXT.AckRequired := FALSE;
   STATUS[789].EXT.Maintanence := FALSE;
   STATUS[789].EXT.Operation := FALSE;
   STATUS[789].EXT.Forced := FALSE;
   STATUS[789].EXT.BIT29 := FALSE;
   STATUS[789].EXT.BIT30 := FALSE;
   STATUS[789].EXT.BIT31 := FALSE;
   STATUS[789].EXT.ModeBit1 := FALSE;
   STATUS[789].EXT.ModeBit2 := FALSE;
   STATUS[789].EXT.ModeBit3 := FALSE;
   STATUS[789].EXT.BIT19 := FALSE;
   STATUS[789].EXT.BIT20 := FALSE;
   STATUS[789].EXT.AlarmSuppressed := FALSE;
   STATUS[789].EXT.AlarmPresent := FALSE;
   STATUS[789].EXT.AlarmFailUnAck := FALSE;
   STATUS[789].Status := 0;
   STATUS[789].TimeStamp := 16#0000;
   STATUS[790].EXT.AlarmWarnUnAck := FALSE;
   STATUS[790].EXT.AckRequired := FALSE;
   STATUS[790].EXT.Maintanence := FALSE;
   STATUS[790].EXT.Operation := FALSE;
   STATUS[790].EXT.Forced := FALSE;
   STATUS[790].EXT.BIT29 := FALSE;
   STATUS[790].EXT.BIT30 := FALSE;
   STATUS[790].EXT.BIT31 := FALSE;
   STATUS[790].EXT.ModeBit1 := FALSE;
   STATUS[790].EXT.ModeBit2 := FALSE;
   STATUS[790].EXT.ModeBit3 := FALSE;
   STATUS[790].EXT.BIT19 := FALSE;
   STATUS[790].EXT.BIT20 := FALSE;
   STATUS[790].EXT.AlarmSuppressed := FALSE;
   STATUS[790].EXT.AlarmPresent := FALSE;
   STATUS[790].EXT.AlarmFailUnAck := FALSE;
   STATUS[790].Status := 0;
   STATUS[790].TimeStamp := 16#0000;
   STATUS[791].EXT.AlarmWarnUnAck := FALSE;
   STATUS[791].EXT.AckRequired := FALSE;
   STATUS[791].EXT.Maintanence := FALSE;
   STATUS[791].EXT.Operation := FALSE;
   STATUS[791].EXT.Forced := FALSE;
   STATUS[791].EXT.BIT29 := FALSE;
   STATUS[791].EXT.BIT30 := FALSE;
   STATUS[791].EXT.BIT31 := FALSE;
   STATUS[791].EXT.ModeBit1 := FALSE;
   STATUS[791].EXT.ModeBit2 := FALSE;
   STATUS[791].EXT.ModeBit3 := FALSE;
   STATUS[791].EXT.BIT19 := FALSE;
   STATUS[791].EXT.BIT20 := FALSE;
   STATUS[791].EXT.AlarmSuppressed := FALSE;
   STATUS[791].EXT.AlarmPresent := FALSE;
   STATUS[791].EXT.AlarmFailUnAck := FALSE;
   STATUS[791].Status := 0;
   STATUS[791].TimeStamp := 16#0000;
   STATUS[792].EXT.AlarmWarnUnAck := FALSE;
   STATUS[792].EXT.AckRequired := FALSE;
   STATUS[792].EXT.Maintanence := FALSE;
   STATUS[792].EXT.Operation := FALSE;
   STATUS[792].EXT.Forced := FALSE;
   STATUS[792].EXT.BIT29 := FALSE;
   STATUS[792].EXT.BIT30 := FALSE;
   STATUS[792].EXT.BIT31 := FALSE;
   STATUS[792].EXT.ModeBit1 := FALSE;
   STATUS[792].EXT.ModeBit2 := FALSE;
   STATUS[792].EXT.ModeBit3 := FALSE;
   STATUS[792].EXT.BIT19 := FALSE;
   STATUS[792].EXT.BIT20 := FALSE;
   STATUS[792].EXT.AlarmSuppressed := FALSE;
   STATUS[792].EXT.AlarmPresent := FALSE;
   STATUS[792].EXT.AlarmFailUnAck := FALSE;
   STATUS[792].Status := 0;
   STATUS[792].TimeStamp := 16#0000;
   STATUS[793].EXT.AlarmWarnUnAck := FALSE;
   STATUS[793].EXT.AckRequired := FALSE;
   STATUS[793].EXT.Maintanence := FALSE;
   STATUS[793].EXT.Operation := FALSE;
   STATUS[793].EXT.Forced := FALSE;
   STATUS[793].EXT.BIT29 := FALSE;
   STATUS[793].EXT.BIT30 := FALSE;
   STATUS[793].EXT.BIT31 := FALSE;
   STATUS[793].EXT.ModeBit1 := FALSE;
   STATUS[793].EXT.ModeBit2 := FALSE;
   STATUS[793].EXT.ModeBit3 := FALSE;
   STATUS[793].EXT.BIT19 := FALSE;
   STATUS[793].EXT.BIT20 := FALSE;
   STATUS[793].EXT.AlarmSuppressed := FALSE;
   STATUS[793].EXT.AlarmPresent := FALSE;
   STATUS[793].EXT.AlarmFailUnAck := FALSE;
   STATUS[793].Status := 0;
   STATUS[793].TimeStamp := 16#0000;
   STATUS[794].EXT.AlarmWarnUnAck := FALSE;
   STATUS[794].EXT.AckRequired := FALSE;
   STATUS[794].EXT.Maintanence := FALSE;
   STATUS[794].EXT.Operation := FALSE;
   STATUS[794].EXT.Forced := FALSE;
   STATUS[794].EXT.BIT29 := FALSE;
   STATUS[794].EXT.BIT30 := FALSE;
   STATUS[794].EXT.BIT31 := FALSE;
   STATUS[794].EXT.ModeBit1 := FALSE;
   STATUS[794].EXT.ModeBit2 := FALSE;
   STATUS[794].EXT.ModeBit3 := FALSE;
   STATUS[794].EXT.BIT19 := FALSE;
   STATUS[794].EXT.BIT20 := FALSE;
   STATUS[794].EXT.AlarmSuppressed := FALSE;
   STATUS[794].EXT.AlarmPresent := FALSE;
   STATUS[794].EXT.AlarmFailUnAck := FALSE;
   STATUS[794].Status := 0;
   STATUS[794].TimeStamp := 16#0000;
   STATUS[795].EXT.AlarmWarnUnAck := FALSE;
   STATUS[795].EXT.AckRequired := FALSE;
   STATUS[795].EXT.Maintanence := FALSE;
   STATUS[795].EXT.Operation := FALSE;
   STATUS[795].EXT.Forced := FALSE;
   STATUS[795].EXT.BIT29 := FALSE;
   STATUS[795].EXT.BIT30 := FALSE;
   STATUS[795].EXT.BIT31 := FALSE;
   STATUS[795].EXT.ModeBit1 := FALSE;
   STATUS[795].EXT.ModeBit2 := FALSE;
   STATUS[795].EXT.ModeBit3 := FALSE;
   STATUS[795].EXT.BIT19 := FALSE;
   STATUS[795].EXT.BIT20 := FALSE;
   STATUS[795].EXT.AlarmSuppressed := FALSE;
   STATUS[795].EXT.AlarmPresent := FALSE;
   STATUS[795].EXT.AlarmFailUnAck := FALSE;
   STATUS[795].Status := 0;
   STATUS[795].TimeStamp := 16#0000;
   STATUS[796].EXT.AlarmWarnUnAck := FALSE;
   STATUS[796].EXT.AckRequired := FALSE;
   STATUS[796].EXT.Maintanence := FALSE;
   STATUS[796].EXT.Operation := FALSE;
   STATUS[796].EXT.Forced := FALSE;
   STATUS[796].EXT.BIT29 := FALSE;
   STATUS[796].EXT.BIT30 := FALSE;
   STATUS[796].EXT.BIT31 := FALSE;
   STATUS[796].EXT.ModeBit1 := FALSE;
   STATUS[796].EXT.ModeBit2 := FALSE;
   STATUS[796].EXT.ModeBit3 := FALSE;
   STATUS[796].EXT.BIT19 := FALSE;
   STATUS[796].EXT.BIT20 := FALSE;
   STATUS[796].EXT.AlarmSuppressed := FALSE;
   STATUS[796].EXT.AlarmPresent := FALSE;
   STATUS[796].EXT.AlarmFailUnAck := FALSE;
   STATUS[796].Status := 0;
   STATUS[796].TimeStamp := 16#0000;
   STATUS[797].EXT.AlarmWarnUnAck := FALSE;
   STATUS[797].EXT.AckRequired := FALSE;
   STATUS[797].EXT.Maintanence := FALSE;
   STATUS[797].EXT.Operation := FALSE;
   STATUS[797].EXT.Forced := FALSE;
   STATUS[797].EXT.BIT29 := FALSE;
   STATUS[797].EXT.BIT30 := FALSE;
   STATUS[797].EXT.BIT31 := FALSE;
   STATUS[797].EXT.ModeBit1 := FALSE;
   STATUS[797].EXT.ModeBit2 := FALSE;
   STATUS[797].EXT.ModeBit3 := FALSE;
   STATUS[797].EXT.BIT19 := FALSE;
   STATUS[797].EXT.BIT20 := FALSE;
   STATUS[797].EXT.AlarmSuppressed := FALSE;
   STATUS[797].EXT.AlarmPresent := FALSE;
   STATUS[797].EXT.AlarmFailUnAck := FALSE;
   STATUS[797].Status := 0;
   STATUS[797].TimeStamp := 16#0000;
   STATUS[798].EXT.AlarmWarnUnAck := FALSE;
   STATUS[798].EXT.AckRequired := FALSE;
   STATUS[798].EXT.Maintanence := FALSE;
   STATUS[798].EXT.Operation := FALSE;
   STATUS[798].EXT.Forced := FALSE;
   STATUS[798].EXT.BIT29 := FALSE;
   STATUS[798].EXT.BIT30 := FALSE;
   STATUS[798].EXT.BIT31 := FALSE;
   STATUS[798].EXT.ModeBit1 := FALSE;
   STATUS[798].EXT.ModeBit2 := FALSE;
   STATUS[798].EXT.ModeBit3 := FALSE;
   STATUS[798].EXT.BIT19 := FALSE;
   STATUS[798].EXT.BIT20 := FALSE;
   STATUS[798].EXT.AlarmSuppressed := FALSE;
   STATUS[798].EXT.AlarmPresent := FALSE;
   STATUS[798].EXT.AlarmFailUnAck := FALSE;
   STATUS[798].Status := 0;
   STATUS[798].TimeStamp := 16#0000;
   STATUS[799].EXT.AlarmWarnUnAck := FALSE;
   STATUS[799].EXT.AckRequired := FALSE;
   STATUS[799].EXT.Maintanence := FALSE;
   STATUS[799].EXT.Operation := FALSE;
   STATUS[799].EXT.Forced := FALSE;
   STATUS[799].EXT.BIT29 := FALSE;
   STATUS[799].EXT.BIT30 := FALSE;
   STATUS[799].EXT.BIT31 := FALSE;
   STATUS[799].EXT.ModeBit1 := FALSE;
   STATUS[799].EXT.ModeBit2 := FALSE;
   STATUS[799].EXT.ModeBit3 := FALSE;
   STATUS[799].EXT.BIT19 := FALSE;
   STATUS[799].EXT.BIT20 := FALSE;
   STATUS[799].EXT.AlarmSuppressed := FALSE;
   STATUS[799].EXT.AlarmPresent := FALSE;
   STATUS[799].EXT.AlarmFailUnAck := FALSE;
   STATUS[799].Status := 0;
   STATUS[799].TimeStamp := 16#0000;
   STATUS[800].EXT.AlarmWarnUnAck := FALSE;
   STATUS[800].EXT.AckRequired := FALSE;
   STATUS[800].EXT.Maintanence := FALSE;
   STATUS[800].EXT.Operation := FALSE;
   STATUS[800].EXT.Forced := FALSE;
   STATUS[800].EXT.BIT29 := FALSE;
   STATUS[800].EXT.BIT30 := FALSE;
   STATUS[800].EXT.BIT31 := FALSE;
   STATUS[800].EXT.ModeBit1 := FALSE;
   STATUS[800].EXT.ModeBit2 := FALSE;
   STATUS[800].EXT.ModeBit3 := FALSE;
   STATUS[800].EXT.BIT19 := FALSE;
   STATUS[800].EXT.BIT20 := FALSE;
   STATUS[800].EXT.AlarmSuppressed := FALSE;
   STATUS[800].EXT.AlarmPresent := FALSE;
   STATUS[800].EXT.AlarmFailUnAck := FALSE;
   STATUS[800].Status := 0;
   STATUS[800].TimeStamp := 16#0000;
   STATUS[801].EXT.AlarmWarnUnAck := FALSE;
   STATUS[801].EXT.AckRequired := FALSE;
   STATUS[801].EXT.Maintanence := FALSE;
   STATUS[801].EXT.Operation := FALSE;
   STATUS[801].EXT.Forced := FALSE;
   STATUS[801].EXT.BIT29 := FALSE;
   STATUS[801].EXT.BIT30 := FALSE;
   STATUS[801].EXT.BIT31 := FALSE;
   STATUS[801].EXT.ModeBit1 := FALSE;
   STATUS[801].EXT.ModeBit2 := FALSE;
   STATUS[801].EXT.ModeBit3 := FALSE;
   STATUS[801].EXT.BIT19 := FALSE;
   STATUS[801].EXT.BIT20 := FALSE;
   STATUS[801].EXT.AlarmSuppressed := FALSE;
   STATUS[801].EXT.AlarmPresent := FALSE;
   STATUS[801].EXT.AlarmFailUnAck := FALSE;
   STATUS[801].Status := 0;
   STATUS[801].TimeStamp := 16#0000;
   STATUS[802].EXT.AlarmWarnUnAck := FALSE;
   STATUS[802].EXT.AckRequired := FALSE;
   STATUS[802].EXT.Maintanence := FALSE;
   STATUS[802].EXT.Operation := FALSE;
   STATUS[802].EXT.Forced := FALSE;
   STATUS[802].EXT.BIT29 := FALSE;
   STATUS[802].EXT.BIT30 := FALSE;
   STATUS[802].EXT.BIT31 := FALSE;
   STATUS[802].EXT.ModeBit1 := FALSE;
   STATUS[802].EXT.ModeBit2 := FALSE;
   STATUS[802].EXT.ModeBit3 := FALSE;
   STATUS[802].EXT.BIT19 := FALSE;
   STATUS[802].EXT.BIT20 := FALSE;
   STATUS[802].EXT.AlarmSuppressed := FALSE;
   STATUS[802].EXT.AlarmPresent := FALSE;
   STATUS[802].EXT.AlarmFailUnAck := FALSE;
   STATUS[802].Status := 0;
   STATUS[802].TimeStamp := 16#0000;
   STATUS[803].EXT.AlarmWarnUnAck := FALSE;
   STATUS[803].EXT.AckRequired := FALSE;
   STATUS[803].EXT.Maintanence := FALSE;
   STATUS[803].EXT.Operation := FALSE;
   STATUS[803].EXT.Forced := FALSE;
   STATUS[803].EXT.BIT29 := FALSE;
   STATUS[803].EXT.BIT30 := FALSE;
   STATUS[803].EXT.BIT31 := FALSE;
   STATUS[803].EXT.ModeBit1 := FALSE;
   STATUS[803].EXT.ModeBit2 := FALSE;
   STATUS[803].EXT.ModeBit3 := FALSE;
   STATUS[803].EXT.BIT19 := FALSE;
   STATUS[803].EXT.BIT20 := FALSE;
   STATUS[803].EXT.AlarmSuppressed := FALSE;
   STATUS[803].EXT.AlarmPresent := FALSE;
   STATUS[803].EXT.AlarmFailUnAck := FALSE;
   STATUS[803].Status := 0;
   STATUS[803].TimeStamp := 16#0000;
   STATUS[804].EXT.AlarmWarnUnAck := FALSE;
   STATUS[804].EXT.AckRequired := FALSE;
   STATUS[804].EXT.Maintanence := FALSE;
   STATUS[804].EXT.Operation := FALSE;
   STATUS[804].EXT.Forced := FALSE;
   STATUS[804].EXT.BIT29 := FALSE;
   STATUS[804].EXT.BIT30 := FALSE;
   STATUS[804].EXT.BIT31 := FALSE;
   STATUS[804].EXT.ModeBit1 := FALSE;
   STATUS[804].EXT.ModeBit2 := FALSE;
   STATUS[804].EXT.ModeBit3 := FALSE;
   STATUS[804].EXT.BIT19 := FALSE;
   STATUS[804].EXT.BIT20 := FALSE;
   STATUS[804].EXT.AlarmSuppressed := FALSE;
   STATUS[804].EXT.AlarmPresent := FALSE;
   STATUS[804].EXT.AlarmFailUnAck := FALSE;
   STATUS[804].Status := 0;
   STATUS[804].TimeStamp := 16#0000;
   STATUS[805].EXT.AlarmWarnUnAck := FALSE;
   STATUS[805].EXT.AckRequired := FALSE;
   STATUS[805].EXT.Maintanence := FALSE;
   STATUS[805].EXT.Operation := FALSE;
   STATUS[805].EXT.Forced := FALSE;
   STATUS[805].EXT.BIT29 := FALSE;
   STATUS[805].EXT.BIT30 := FALSE;
   STATUS[805].EXT.BIT31 := FALSE;
   STATUS[805].EXT.ModeBit1 := FALSE;
   STATUS[805].EXT.ModeBit2 := FALSE;
   STATUS[805].EXT.ModeBit3 := FALSE;
   STATUS[805].EXT.BIT19 := FALSE;
   STATUS[805].EXT.BIT20 := FALSE;
   STATUS[805].EXT.AlarmSuppressed := FALSE;
   STATUS[805].EXT.AlarmPresent := FALSE;
   STATUS[805].EXT.AlarmFailUnAck := FALSE;
   STATUS[805].Status := 0;
   STATUS[805].TimeStamp := 16#0000;
   STATUS[806].EXT.AlarmWarnUnAck := FALSE;
   STATUS[806].EXT.AckRequired := FALSE;
   STATUS[806].EXT.Maintanence := FALSE;
   STATUS[806].EXT.Operation := FALSE;
   STATUS[806].EXT.Forced := FALSE;
   STATUS[806].EXT.BIT29 := FALSE;
   STATUS[806].EXT.BIT30 := FALSE;
   STATUS[806].EXT.BIT31 := FALSE;
   STATUS[806].EXT.ModeBit1 := FALSE;
   STATUS[806].EXT.ModeBit2 := FALSE;
   STATUS[806].EXT.ModeBit3 := FALSE;
   STATUS[806].EXT.BIT19 := FALSE;
   STATUS[806].EXT.BIT20 := FALSE;
   STATUS[806].EXT.AlarmSuppressed := FALSE;
   STATUS[806].EXT.AlarmPresent := FALSE;
   STATUS[806].EXT.AlarmFailUnAck := FALSE;
   STATUS[806].Status := 0;
   STATUS[806].TimeStamp := 16#0000;
   STATUS[807].EXT.AlarmWarnUnAck := FALSE;
   STATUS[807].EXT.AckRequired := FALSE;
   STATUS[807].EXT.Maintanence := FALSE;
   STATUS[807].EXT.Operation := FALSE;
   STATUS[807].EXT.Forced := FALSE;
   STATUS[807].EXT.BIT29 := FALSE;
   STATUS[807].EXT.BIT30 := FALSE;
   STATUS[807].EXT.BIT31 := FALSE;
   STATUS[807].EXT.ModeBit1 := FALSE;
   STATUS[807].EXT.ModeBit2 := FALSE;
   STATUS[807].EXT.ModeBit3 := FALSE;
   STATUS[807].EXT.BIT19 := FALSE;
   STATUS[807].EXT.BIT20 := FALSE;
   STATUS[807].EXT.AlarmSuppressed := FALSE;
   STATUS[807].EXT.AlarmPresent := FALSE;
   STATUS[807].EXT.AlarmFailUnAck := FALSE;
   STATUS[807].Status := 0;
   STATUS[807].TimeStamp := 16#0000;
   STATUS[808].EXT.AlarmWarnUnAck := FALSE;
   STATUS[808].EXT.AckRequired := FALSE;
   STATUS[808].EXT.Maintanence := FALSE;
   STATUS[808].EXT.Operation := FALSE;
   STATUS[808].EXT.Forced := FALSE;
   STATUS[808].EXT.BIT29 := FALSE;
   STATUS[808].EXT.BIT30 := FALSE;
   STATUS[808].EXT.BIT31 := FALSE;
   STATUS[808].EXT.ModeBit1 := FALSE;
   STATUS[808].EXT.ModeBit2 := FALSE;
   STATUS[808].EXT.ModeBit3 := FALSE;
   STATUS[808].EXT.BIT19 := FALSE;
   STATUS[808].EXT.BIT20 := FALSE;
   STATUS[808].EXT.AlarmSuppressed := FALSE;
   STATUS[808].EXT.AlarmPresent := FALSE;
   STATUS[808].EXT.AlarmFailUnAck := FALSE;
   STATUS[808].Status := 0;
   STATUS[808].TimeStamp := 16#0000;
   STATUS[809].EXT.AlarmWarnUnAck := FALSE;
   STATUS[809].EXT.AckRequired := FALSE;
   STATUS[809].EXT.Maintanence := FALSE;
   STATUS[809].EXT.Operation := FALSE;
   STATUS[809].EXT.Forced := FALSE;
   STATUS[809].EXT.BIT29 := FALSE;
   STATUS[809].EXT.BIT30 := FALSE;
   STATUS[809].EXT.BIT31 := FALSE;
   STATUS[809].EXT.ModeBit1 := FALSE;
   STATUS[809].EXT.ModeBit2 := FALSE;
   STATUS[809].EXT.ModeBit3 := FALSE;
   STATUS[809].EXT.BIT19 := FALSE;
   STATUS[809].EXT.BIT20 := FALSE;
   STATUS[809].EXT.AlarmSuppressed := FALSE;
   STATUS[809].EXT.AlarmPresent := FALSE;
   STATUS[809].EXT.AlarmFailUnAck := FALSE;
   STATUS[809].Status := 0;
   STATUS[809].TimeStamp := 16#0000;
   STATUS[810].EXT.AlarmWarnUnAck := FALSE;
   STATUS[810].EXT.AckRequired := FALSE;
   STATUS[810].EXT.Maintanence := FALSE;
   STATUS[810].EXT.Operation := FALSE;
   STATUS[810].EXT.Forced := FALSE;
   STATUS[810].EXT.BIT29 := FALSE;
   STATUS[810].EXT.BIT30 := FALSE;
   STATUS[810].EXT.BIT31 := FALSE;
   STATUS[810].EXT.ModeBit1 := FALSE;
   STATUS[810].EXT.ModeBit2 := FALSE;
   STATUS[810].EXT.ModeBit3 := FALSE;
   STATUS[810].EXT.BIT19 := FALSE;
   STATUS[810].EXT.BIT20 := FALSE;
   STATUS[810].EXT.AlarmSuppressed := FALSE;
   STATUS[810].EXT.AlarmPresent := FALSE;
   STATUS[810].EXT.AlarmFailUnAck := FALSE;
   STATUS[810].Status := 0;
   STATUS[810].TimeStamp := 16#0000;
   STATUS[811].EXT.AlarmWarnUnAck := FALSE;
   STATUS[811].EXT.AckRequired := FALSE;
   STATUS[811].EXT.Maintanence := FALSE;
   STATUS[811].EXT.Operation := FALSE;
   STATUS[811].EXT.Forced := FALSE;
   STATUS[811].EXT.BIT29 := FALSE;
   STATUS[811].EXT.BIT30 := FALSE;
   STATUS[811].EXT.BIT31 := FALSE;
   STATUS[811].EXT.ModeBit1 := FALSE;
   STATUS[811].EXT.ModeBit2 := FALSE;
   STATUS[811].EXT.ModeBit3 := FALSE;
   STATUS[811].EXT.BIT19 := FALSE;
   STATUS[811].EXT.BIT20 := FALSE;
   STATUS[811].EXT.AlarmSuppressed := FALSE;
   STATUS[811].EXT.AlarmPresent := FALSE;
   STATUS[811].EXT.AlarmFailUnAck := FALSE;
   STATUS[811].Status := 0;
   STATUS[811].TimeStamp := 16#0000;
   STATUS[812].EXT.AlarmWarnUnAck := FALSE;
   STATUS[812].EXT.AckRequired := FALSE;
   STATUS[812].EXT.Maintanence := FALSE;
   STATUS[812].EXT.Operation := FALSE;
   STATUS[812].EXT.Forced := FALSE;
   STATUS[812].EXT.BIT29 := FALSE;
   STATUS[812].EXT.BIT30 := FALSE;
   STATUS[812].EXT.BIT31 := FALSE;
   STATUS[812].EXT.ModeBit1 := FALSE;
   STATUS[812].EXT.ModeBit2 := FALSE;
   STATUS[812].EXT.ModeBit3 := FALSE;
   STATUS[812].EXT.BIT19 := FALSE;
   STATUS[812].EXT.BIT20 := FALSE;
   STATUS[812].EXT.AlarmSuppressed := FALSE;
   STATUS[812].EXT.AlarmPresent := FALSE;
   STATUS[812].EXT.AlarmFailUnAck := FALSE;
   STATUS[812].Status := 0;
   STATUS[812].TimeStamp := 16#0000;
   STATUS[813].EXT.AlarmWarnUnAck := FALSE;
   STATUS[813].EXT.AckRequired := FALSE;
   STATUS[813].EXT.Maintanence := FALSE;
   STATUS[813].EXT.Operation := FALSE;
   STATUS[813].EXT.Forced := FALSE;
   STATUS[813].EXT.BIT29 := FALSE;
   STATUS[813].EXT.BIT30 := FALSE;
   STATUS[813].EXT.BIT31 := FALSE;
   STATUS[813].EXT.ModeBit1 := FALSE;
   STATUS[813].EXT.ModeBit2 := FALSE;
   STATUS[813].EXT.ModeBit3 := FALSE;
   STATUS[813].EXT.BIT19 := FALSE;
   STATUS[813].EXT.BIT20 := FALSE;
   STATUS[813].EXT.AlarmSuppressed := FALSE;
   STATUS[813].EXT.AlarmPresent := FALSE;
   STATUS[813].EXT.AlarmFailUnAck := FALSE;
   STATUS[813].Status := 0;
   STATUS[813].TimeStamp := 16#0000;
   STATUS[814].EXT.AlarmWarnUnAck := FALSE;
   STATUS[814].EXT.AckRequired := FALSE;
   STATUS[814].EXT.Maintanence := FALSE;
   STATUS[814].EXT.Operation := FALSE;
   STATUS[814].EXT.Forced := FALSE;
   STATUS[814].EXT.BIT29 := FALSE;
   STATUS[814].EXT.BIT30 := FALSE;
   STATUS[814].EXT.BIT31 := FALSE;
   STATUS[814].EXT.ModeBit1 := FALSE;
   STATUS[814].EXT.ModeBit2 := FALSE;
   STATUS[814].EXT.ModeBit3 := FALSE;
   STATUS[814].EXT.BIT19 := FALSE;
   STATUS[814].EXT.BIT20 := FALSE;
   STATUS[814].EXT.AlarmSuppressed := FALSE;
   STATUS[814].EXT.AlarmPresent := FALSE;
   STATUS[814].EXT.AlarmFailUnAck := FALSE;
   STATUS[814].Status := 0;
   STATUS[814].TimeStamp := 16#0000;
   STATUS[815].EXT.AlarmWarnUnAck := FALSE;
   STATUS[815].EXT.AckRequired := FALSE;
   STATUS[815].EXT.Maintanence := FALSE;
   STATUS[815].EXT.Operation := FALSE;
   STATUS[815].EXT.Forced := FALSE;
   STATUS[815].EXT.BIT29 := FALSE;
   STATUS[815].EXT.BIT30 := FALSE;
   STATUS[815].EXT.BIT31 := FALSE;
   STATUS[815].EXT.ModeBit1 := FALSE;
   STATUS[815].EXT.ModeBit2 := FALSE;
   STATUS[815].EXT.ModeBit3 := FALSE;
   STATUS[815].EXT.BIT19 := FALSE;
   STATUS[815].EXT.BIT20 := FALSE;
   STATUS[815].EXT.AlarmSuppressed := FALSE;
   STATUS[815].EXT.AlarmPresent := FALSE;
   STATUS[815].EXT.AlarmFailUnAck := FALSE;
   STATUS[815].Status := 0;
   STATUS[815].TimeStamp := 16#0000;
   STATUS[816].EXT.AlarmWarnUnAck := FALSE;
   STATUS[816].EXT.AckRequired := FALSE;
   STATUS[816].EXT.Maintanence := FALSE;
   STATUS[816].EXT.Operation := FALSE;
   STATUS[816].EXT.Forced := FALSE;
   STATUS[816].EXT.BIT29 := FALSE;
   STATUS[816].EXT.BIT30 := FALSE;
   STATUS[816].EXT.BIT31 := FALSE;
   STATUS[816].EXT.ModeBit1 := FALSE;
   STATUS[816].EXT.ModeBit2 := FALSE;
   STATUS[816].EXT.ModeBit3 := FALSE;
   STATUS[816].EXT.BIT19 := FALSE;
   STATUS[816].EXT.BIT20 := FALSE;
   STATUS[816].EXT.AlarmSuppressed := FALSE;
   STATUS[816].EXT.AlarmPresent := FALSE;
   STATUS[816].EXT.AlarmFailUnAck := FALSE;
   STATUS[816].Status := 0;
   STATUS[816].TimeStamp := 16#0000;
   STATUS[817].EXT.AlarmWarnUnAck := FALSE;
   STATUS[817].EXT.AckRequired := FALSE;
   STATUS[817].EXT.Maintanence := FALSE;
   STATUS[817].EXT.Operation := FALSE;
   STATUS[817].EXT.Forced := FALSE;
   STATUS[817].EXT.BIT29 := FALSE;
   STATUS[817].EXT.BIT30 := FALSE;
   STATUS[817].EXT.BIT31 := FALSE;
   STATUS[817].EXT.ModeBit1 := FALSE;
   STATUS[817].EXT.ModeBit2 := FALSE;
   STATUS[817].EXT.ModeBit3 := FALSE;
   STATUS[817].EXT.BIT19 := FALSE;
   STATUS[817].EXT.BIT20 := FALSE;
   STATUS[817].EXT.AlarmSuppressed := FALSE;
   STATUS[817].EXT.AlarmPresent := FALSE;
   STATUS[817].EXT.AlarmFailUnAck := FALSE;
   STATUS[817].Status := 0;
   STATUS[817].TimeStamp := 16#0000;
   STATUS[818].EXT.AlarmWarnUnAck := FALSE;
   STATUS[818].EXT.AckRequired := FALSE;
   STATUS[818].EXT.Maintanence := FALSE;
   STATUS[818].EXT.Operation := FALSE;
   STATUS[818].EXT.Forced := FALSE;
   STATUS[818].EXT.BIT29 := FALSE;
   STATUS[818].EXT.BIT30 := FALSE;
   STATUS[818].EXT.BIT31 := FALSE;
   STATUS[818].EXT.ModeBit1 := FALSE;
   STATUS[818].EXT.ModeBit2 := FALSE;
   STATUS[818].EXT.ModeBit3 := FALSE;
   STATUS[818].EXT.BIT19 := FALSE;
   STATUS[818].EXT.BIT20 := FALSE;
   STATUS[818].EXT.AlarmSuppressed := FALSE;
   STATUS[818].EXT.AlarmPresent := FALSE;
   STATUS[818].EXT.AlarmFailUnAck := FALSE;
   STATUS[818].Status := 0;
   STATUS[818].TimeStamp := 16#0000;
   STATUS[819].EXT.AlarmWarnUnAck := FALSE;
   STATUS[819].EXT.AckRequired := FALSE;
   STATUS[819].EXT.Maintanence := FALSE;
   STATUS[819].EXT.Operation := FALSE;
   STATUS[819].EXT.Forced := FALSE;
   STATUS[819].EXT.BIT29 := FALSE;
   STATUS[819].EXT.BIT30 := FALSE;
   STATUS[819].EXT.BIT31 := FALSE;
   STATUS[819].EXT.ModeBit1 := FALSE;
   STATUS[819].EXT.ModeBit2 := FALSE;
   STATUS[819].EXT.ModeBit3 := FALSE;
   STATUS[819].EXT.BIT19 := FALSE;
   STATUS[819].EXT.BIT20 := FALSE;
   STATUS[819].EXT.AlarmSuppressed := FALSE;
   STATUS[819].EXT.AlarmPresent := FALSE;
   STATUS[819].EXT.AlarmFailUnAck := FALSE;
   STATUS[819].Status := 0;
   STATUS[819].TimeStamp := 16#0000;
   STATUS[820].EXT.AlarmWarnUnAck := FALSE;
   STATUS[820].EXT.AckRequired := FALSE;
   STATUS[820].EXT.Maintanence := FALSE;
   STATUS[820].EXT.Operation := FALSE;
   STATUS[820].EXT.Forced := FALSE;
   STATUS[820].EXT.BIT29 := FALSE;
   STATUS[820].EXT.BIT30 := FALSE;
   STATUS[820].EXT.BIT31 := FALSE;
   STATUS[820].EXT.ModeBit1 := FALSE;
   STATUS[820].EXT.ModeBit2 := FALSE;
   STATUS[820].EXT.ModeBit3 := FALSE;
   STATUS[820].EXT.BIT19 := FALSE;
   STATUS[820].EXT.BIT20 := FALSE;
   STATUS[820].EXT.AlarmSuppressed := FALSE;
   STATUS[820].EXT.AlarmPresent := FALSE;
   STATUS[820].EXT.AlarmFailUnAck := FALSE;
   STATUS[820].Status := 0;
   STATUS[820].TimeStamp := 16#0000;
   STATUS[821].EXT.AlarmWarnUnAck := FALSE;
   STATUS[821].EXT.AckRequired := FALSE;
   STATUS[821].EXT.Maintanence := FALSE;
   STATUS[821].EXT.Operation := FALSE;
   STATUS[821].EXT.Forced := FALSE;
   STATUS[821].EXT.BIT29 := FALSE;
   STATUS[821].EXT.BIT30 := FALSE;
   STATUS[821].EXT.BIT31 := FALSE;
   STATUS[821].EXT.ModeBit1 := FALSE;
   STATUS[821].EXT.ModeBit2 := FALSE;
   STATUS[821].EXT.ModeBit3 := FALSE;
   STATUS[821].EXT.BIT19 := FALSE;
   STATUS[821].EXT.BIT20 := FALSE;
   STATUS[821].EXT.AlarmSuppressed := FALSE;
   STATUS[821].EXT.AlarmPresent := FALSE;
   STATUS[821].EXT.AlarmFailUnAck := FALSE;
   STATUS[821].Status := 0;
   STATUS[821].TimeStamp := 16#0000;
   STATUS[822].EXT.AlarmWarnUnAck := FALSE;
